// POUs/BACnet Helper/[internal]/_F_BACnet_Utf8ToWin1252
FUNCTION _F_BACnet_Utf8ToWin1252 : BYTE
VAR_INPUT
	pUtf8	: POINTER TO BYTE;
	cbUtf8	: UDINT; (* byte size of UTF8 character (1...6) *)
END_VAR
VAR
	pArr		: POINTER TO ARRAY[0..5] OF BYTE;
	pWord		: POINTER TO ARRAY[0..1] OF BYTE;
	wUCS2		: WORD;
END_VAR
VAR CONSTANT
	cRepl	: BYTE := 16#5F;
END_VAR

(*
	Windows-Codepages
874		Thai
932		Japanisch
936		Vereinfachtes Chinesisch
949		Koreanisch
950		Traditionelles Chinesisch
1250	Mitteleuropäisch
1251	Kyrillisch
1252	Westeuropäisch
1253	Griechisch
1254	Türkisch
1255	Hebräisch
1256	Arabisch
1257	Baltisch
1258	Vietnamesisch
*)
(* first step - convert to UCS2 *)
pArr := pUtf8;
IF (pArr^[0] <= 16#7F) THEN
	(* basic latin *)
	_F_BACnet_Utf8ToWin1252 := pArr^[0];
	RETURN;
ELSIF (cbUtf8 >= 2) THEN
	pWord := ADR(wUCS2);
	IF (pArr^[0] = 16#C2) THEN
		(* latin-1 supplement *)
		wUCS2 := pArr^[1];
	ELSIF (pArr^[0] = 16#C3) AND (pArr^[1] <= 16#BF) THEN
		(* latin-1 supplement *)
		wUCS2 := pArr^[1] + 16#40;
	ELSIF (pArr^[0] = 16#C4) AND (pArr^[1] >= 16#80) THEN
		(* latin extended-A *)
		pWord^[1] := 16#01;
		pWord^[0] := pArr^[1] - 16#80;
	ELSIF (pArr^[0] = 16#C5) AND (pArr^[1] >= 16#80) THEN
		(* latin extended-A *)
		pWord^[1] := 16#01;
		pWord^[0] := pArr^[1] - 16#40;
	ELSIF (pArr^[0] = 16#C6) AND (pArr^[1] >= 16#80) THEN
		(* latin extended-B *)
		pWord^[1] := 16#01;
		pWord^[0] := pArr^[1];
	ELSIF (pArr^[0] = 16#C7) AND (pArr^[1] <= 16#BF) THEN
		(* latin extended-B *)
		pWord^[1] := 16#01;
		pWord^[0] := pArr^[1] + 16#40;
	ELSIF (cbUtf8 >= 3) THEN
		IF (pArr^[0] = 16#E2) AND (pArr^[1] = 16#82) THEN
			(* currency symbols *)
			pWord^[1] := 16#20;
			pWord^[0] := pArr^[2];
		ELSE
			(* unsupported *)
			_F_BACnet_Utf8ToWin1252 := cRepl;
			RETURN;
		END_IF
	ELSE
		(* unsupported *)
		_F_BACnet_Utf8ToWin1252 := cRepl;
		RETURN;
	END_IF
	(* convert UCS2 to Windows-1252 *)
	_F_BACnet_Utf8ToWin1252 := _F_BACnet_UCS2ToWin1252(pWord, FALSE);
	RETURN;
END_IF
(* unsupported *)
_F_BACnet_Utf8ToWin1252 := cRepl;

END_FUNCTION

// POUs/BACnet Helper/[internal]/_F_BACnet_UCS2ToWin1252
FUNCTION _F_BACnet_UCS2ToWin1252 : BYTE
VAR_INPUT
	pUCS2 :	POINTER TO WORD;
	bBE	: BOOL; (* byte-order big endian = TRUE *)
END_VAR
VAR
	pArr : POINTER TO ARRAY[0..1] OF BYTE;
	wUCS2: WORD;
END_VAR
VAR CONSTANT
	cRepl	: BYTE := 16#5F;
END_VAR

(*
	Windows-Codepages
874		Thai
932		Japanisch
936		Vereinfachtes Chinesisch
949		Koreanisch
950		Traditionelles Chinesisch
1250	Mitteleuropäisch
1251	Kyrillisch
1252	Westeuropäisch
1253	Griechisch
1254	Türkisch
1255	Hebräisch
1256	Arabisch
1257	Baltisch
1258	Vietnamesisch
*)
pArr := pUCS2;
IF bBE THEN
	wUCS2 := (pArr^[0] * 16#0100) + pArr^[1];
ELSE
	wUCS2 := pUCS2^;
END_IF
CASE wUCS2 OF
	16#178: 	_F_BACnet_UCS2ToWin1252 := 16#9F;
	16#153: 	_F_BACnet_UCS2ToWin1252 := 16#9C;
	16#152: 	_F_BACnet_UCS2ToWin1252 := 16#8C;
	16#17E: 	_F_BACnet_UCS2ToWin1252 := 16#9E;
	16#17D: 	_F_BACnet_UCS2ToWin1252 := 16#8E;
	16#161: 	_F_BACnet_UCS2ToWin1252 := 16#9A;
	16#160: 	_F_BACnet_UCS2ToWin1252 := 16#8A;
	16#20AC: 	_F_BACnet_UCS2ToWin1252 := 16#80;
	ELSE
		IF wUCS2 <= 16#FF THEN
			_F_BACnet_UCS2ToWin1252 := WORD_TO_BYTE(wUCS2);
		ELSE
			_F_BACnet_UCS2ToWin1252 := cRepl;
		END_IF
END_CASE

END_FUNCTION

// POUs/BACnet Helper/[internal]/_F_BACnet_DecodeUCS2
FUNCTION _F_BACnet_DecodeUCS2 : UDINT (* result is the new character length of the string *)
VAR_INPUT
	pString		: POINTER TO WORD; (* pointer to UCS2 string beginning *)
	cbString	: UDINT; (* byte size of string (use SIZEOF - don't use LEN) *)
END_VAR
VAR
	i		: UDINT;
	pResult	: POINTER TO BYTE;
	pBy		: POINTER TO WORD;
END_VAR

pResult	:= pString;
pBy		:= pString;
FOR i := 0 TO cbString-1 DO
	pResult^ := _F_BACnet_UCS2ToWin1252(pBy, TRUE);
	pBy := pBy + 2;
	(* end-of-string by character *)
	IF (pResult^ = 16#00) THEN
		EXIT;
	END_IF
	(* next character *)
	pResult := pResult + 1;
	(* end-of-string by length *)
	IF (pBy >= (pString + cbString)) THEN
		EXIT;
	END_IF
END_FOR
pResult^ := 16#00;
_F_BACnet_DecodeUCS2 := pResult - pString;

END_FUNCTION

// POUs/BACnet Helper/[internal]/_F_BACnet_DecodeUCS4
FUNCTION _F_BACnet_DecodeUCS4 : UDINT (* result is the new character length of the string *)
VAR_INPUT
	pString		: POINTER TO DWORD; (* pointer to UCS4 string beginning *)
	cbString	: UDINT; (* byte size of string (use SIZEOF - don't use LEN) *)
END_VAR
VAR
	i		: UDINT;
	pResult	: POINTER TO BYTE;
	pBy		: POINTER TO WORD;
END_VAR

pResult	:= pString;
pBy		:= pString;
FOR i := 0 TO cbString-1 DO
	(* byte order big endian *)
	pResult^ := _F_BACnet_UCS2ToWin1252(pBy+2, TRUE);
	pBy := pBy + 4;
	(* end-of-string by character *)
	IF (pResult^ = 16#00) THEN
		EXIT;
	END_IF
	(* next character *)
	pResult := pResult + 1;
	(* end-of-string by length *)
	IF (pBy >= (pString + cbString)) THEN
		EXIT;
	END_IF
END_FOR
pResult^ := 16#00;
_F_BACnet_DecodeUCS4 := pResult - pString;

END_FUNCTION

// POUs/BACnet ADS/Properties/FB_BACnet_EventMessageTextsProperty
FUNCTION_BLOCK FB_BACnet_EventMessageTextsProperty
VAR_INPUT
	tObjectID			: T_BACnet_ObjectIdentifier := 16#FFFFFFFF;
	bAutoGet			: BOOL:=TRUE; (* TRUE = get data from property when ADS connection OR object ID changed *)
	bGet				: BOOL; (* FALSE --> TRUE = get data from property *)
END_VAR
VAR_IN_OUT
	stAdsConn			: ST_BACnet_AdsConnection;
END_VAR
VAR_OUTPUT
	bDone				: BOOL;
	bBusy				: BOOL;
	bError				: BOOL;
	nErrorId			: UINT;
	arrTexts			: ARRAY[0..2] OF T_MaxString; (* Windows-1252 encoded *)
END_VAR
VAR
	_fbReadProp		: FB_BACnet_ReadProp;
	_i				: INT;
	_rtrigGet		: R_TRIG;

	_iEntry			: INT;
	_pEntry			: POINTER TO ST_BACnet_CharacterStringExtListEntry;
	_pText			: POINTER TO BYTE;
	_pByte			: POINTER TO BYTE;
	_bNextEntry		: BOOL;
	_cbEntrySize	: UDINT;
	_cbTmpSize		: UDINT;
	_cbTotalBuf		: UDINT;
	_nAdsReloadOld	: USINT;
	_tObjectIDOld	: T_BACnet_ObjectIdentifier := 16#FFFFFFFF;
	_strExtDecode	: FB_BACnet_StringExtDecode;

END_VAR

(*

Listheader:

typedef struct _ListEntryHdr
{
      DWORD nEntrySize;
      DWORD hdrInfo;
}ListEntryHdr, *PListEntryHdr;


typedef struct _BACnetCharacterString
{
      ULONG       cookie            : 8; // = 0 -> do differentiate normal strings
      ULONG       encoding          : 8; 
      ULONG       strLen            : 16;
      BYTE        stringData[BACNET_STRING_MAXLENGTH];
}BACnetCharacterString, *PBACnetCharacterString;

#define     BACNET_STRING_MAXLENGTH 256

*)

(* ADS read *)
_fbReadProp(
	BACnetDevicePort	:= stAdsConn.nAmsPort,
	bExecute			:= ,
	sNetId				:= stAdsConn.sAmsNetId,
	ObjectType			:= F_BACnet_GetObjType(tObjectID),
	PropertyID			:= BACnetPropertyIdentifier_EventMessageTexts,
	DataType			:= BACnetDataType_CharacterStringExtList,
	ObjectInstance		:= F_BACnet_GetObjInstance(tObjectID),
	ptrValue			:= ADR(stBACnet_AdsBuffer.arrData),
	nLenValue			:= SIZEOF(stBACnet_AdsBuffer.arrData),
	bDone				=> ,
	bBusy				=> ,
	bError				=> ,
	nErrID				=> ,
	nProcessedLen		=> );

(* trigger start event *)
_rtrigGet(CLK:= bGet, Q=> );

(* state machine *)
CASE _i OF

	0: (* Idle *)
		IF 		_rtrigGet.Q
			OR	(		(		(_nAdsReloadOld <> stAdsConn.nReload)
							OR	(_tObjectIDOld <> tObjectID)
						)
					AND	bAutoGet
				)
		THEN
			IF (NOT stAdsConn.bValid) THEN
				(* ADS connection not valid *)
				nErrorId := BACnet_ERR_INVALID_ADS_CONN;
			ELSIF (NOT stAdsConn.bServer AND NOT stAdsConn.bClient) THEN
				(* not a server nor a client *)
				nErrorId := BACnet_ERR_ADS_NoServerClient;
			ELSE
				_i := 1;
				nErrorId := BACnet_ERR_NO_ERROR;
				(* remind parameter *)
				_tObjectIDOld := tObjectID;
				_nAdsReloadOld := stAdsConn.nReload;
			END_IF
			(* reset done flag *)
			bDone := FALSE;
		END_IF
		IF (NOT bGet) AND (NOT bAutoGet) THEN
			nErrorId := BACnet_ERR_NO_ERROR;
			bDone := FALSE;
		END_IF

	(* READ *)
	1: (* read object property data over ADS *)
		IF TestAndSet(stBACnet_AdsBuffer.bTestSet) THEN
			IF _fbReadProp.bExecute THEN
				IF _fbReadProp.bError THEN
					_i := 100;
					nErrorId := BACnet_ERR_ADS_Read;
					_fbReadProp.bExecute := FALSE;
				ELSIF (NOT _fbReadProp.bBusy) THEN
					_i := 2;
					_fbReadProp.bExecute := FALSE;
					_pEntry := ADR(stBACnet_AdsBuffer.arrData);
					MEMSET(ADR(arrTexts), 0, SIZEOF(arrTexts));
					_cbTotalBuf := 0;
					_iEntry := 0;
				END_IF
			ELSE
				(* lock global ADS buffer and start reading *)
				IF stBACnet_AdsBuffer.iLocked = 0 THEN
					_fbReadProp.bExecute := TRUE;
					stBACnet_AdsBuffer.iLocked := SIZEOF(stBACnet_AdsBuffer.arrData);
				END_IF
			END_IF

			(* release temporary task lock *)
			stBACnet_AdsBuffer.bTestSet := FALSE;
		END_IF

	2: (* select time value *)
		WHILE (_i = 2) DO
			_cbEntrySize := _pEntry^.nEntrySize AND 16#7FFFFFFF;
			(* check entry size *)
			IF (_cbEntrySize) > 0 THEN
				(* check index *)
				IF (_iEntry > 2) THEN
					(* error, too many entries *)
					nErrorId := BACnet_ERR_ADS_TooManyEntries;
					_i := 100;
				ELSE
					(* try to decode property data *)
					_strExtDecode(
						pChrStringExt:= ADR(_pEntry^.extString),
						cbOutSize	:= SIZEOF(arrTexts[_iEntry]),
						pOutString	:= ADR(arrTexts[_iEntry]),
						bValid		=> ,
						bOverflow	=> ,
						bUnsupported=> ,
						nLength		=> ,
						eSrcEncoding=> );
					(* check error flags *)
					IF _strExtDecode.bOverflow THEN
						(* text too long *)
						nErrorId := BACnet_ERR_ADS_WrongEntrySize;
						_i := 100;
					ELSIF _strExtDecode.bUnsupported THEN
						(* unsupported encoding *)
						nErrorId := BACnet_ERR_ADS_Encoding;
						_i := 100;
					END_IF
				END_IF
			END_IF

			(* next entry *)
			_NextEntry();
			_iEntry := _iEntry + 1;

			(* check if next entry available *)
			IF (NOT _bNextEntry) THEN
				IF (_iEntry < 3) THEN
					(* not enough entries *)
					nErrorId := BACnet_ERR_ADS_NotEnoughEntries;
				END_IF
				_i := 100;
			END_IF

		END_WHILE

	100: (* Done *)
		bDone := (nErrorId = BACnet_ERR_NO_ERROR);
		(* release ADS buffer *)
		stBACnet_AdsBuffer.iLocked := 0;
		(* go idle *)
		_i := 0;

END_CASE

(* set error flag *)
bError 	:= nErrorId > BACnet_ERR_NO_ERROR;
bBusy 	:= _i > 0;

ACTION _NextEntry:
_bNextEntry := (_pEntry^.nEntrySize AND 16#80000000) = 16#80000000;
_cbTmpSize := _F_BACnet_AlignedSize((_pEntry^.nEntrySize AND 16#7FFFFFFF) + SIZEOF(_pEntry^.nEntrySize) + SIZEOF(_pEntry^.hdrInfo));
_pEntry := _pEntry + _cbTmpSize;
END_ACTION

END_FUNCTION_BLOCK

// POUs/BACnet Helper/[internal]/_F_BACnet_AlignedSize
FUNCTION _F_BACnet_AlignedSize : DWORD
VAR_INPUT
	n	: DWORD;
END_VAR
VAR
END_VAR

_F_BACnet_AlignedSize := (4*(((n)+3)/4));

END_FUNCTION

// POUs/BACnet ADS/Properties/FB_BACnet_ExceptionScheduleProperty
FUNCTION_BLOCK FB_BACnet_ExceptionScheduleProperty
VAR_INPUT
	tObjectID			: T_BACnet_ObjectIdentifier := 16#FFFFFFFF;
	bAutoGet			: BOOL:=TRUE; (* TRUE = get data from property when ADS connection OR object ID changed *)
	bGet				: BOOL; (* FALSE --> TRUE = get data from property *)
	bSet				: BOOL; (* FALSE --> TRUE = set data into property *)
END_VAR
VAR_IN_OUT
	stExceptSched		: ST_BACnet_ExceptionScheduleBool;
	stAdsConn			: ST_BACnet_AdsConnection;
END_VAR
VAR_OUTPUT
	bDone				: BOOL;
	bBusy				: BOOL;
	bError				: BOOL;
	nErrorId			: UINT;
END_VAR
VAR
	_fbReadProp		: FB_BACnet_ReadProp;
	_fbWriteProp	: FB_BACnet_WriteProp;
	_i				: INT;
	_rtrigGet		: R_TRIG;
	_rtrigSet		: R_TRIG;

	_pOldEventEntrySize		: POINTER TO DWORD;
	_pSpEventCalEntryDate	: POINTER TO ST_BACnet_SpecialEventListCalEntryDate;
	_pSpEventCalEntryRange	: POINTER TO ST_BACnet_SpecialEventListCalEntryRange;
	_pSpEventCalEntryWnD	: POINTER TO ST_BACnet_SpecialEventListCalEntryWnD;
	_pSpEventCalRef			: POINTER TO ST_BACnet_SpecialEventListCalReference;
	_pTimeValue		: POINTER TO ST_BACnet_TimeValueList;
	_pOldTimeValue	: POINTER TO ST_BACnet_TimeValueList;

	_iEntry			: INT;
	_iTv			: INT;

	_bNextEvent		: BOOL;
	_bNextTimeValue	: BOOL;

	_cbTmpSize		: UDINT;
	_cbTotalEntry	: UDINT;
	_cbTotalBuf		: UDINT;
	_nAdsReloadOld	: USINT;
	_tObjectIDOld	: T_BACnet_ObjectIdentifier := 16#FFFFFFFF;

END_VAR

(*

Listheader:

typedef struct _ListEntryHdr
{
      DWORD nEntrySize;
      DWORD hdrInfo;
}ListEntryHdr, *PListEntryHdr;

#define ListAlignedSize(n)         (4*(((n)+3)/4))
#define FirstListEntry(p) ( (p)->nEntrySize == 0 )                          ? NULL:p
#define NextListEntry(p) ( ( ((p)->nEntrySize&0x80000000) == 0 ) ? NULL:(PBYTE)(p) + ( ListAlignedSize((p)->nEntrySize&~(0x80000000)) + sizeof(ListEntryHdr)) ) // +4 da für nEntrySize 4 Byte reserviert sind, HighBit ausmaskieren
#define ElemSize(p) ((p)->nEntrySize&(~0x80000000))
#define AlignedEntrySize(p) (ListAlignedSize((p)->nEntrySize&(~0x80000000)))

###################################################################

PropExceptionSchedule:

enum BACnetSpecialEventChoice
{
      calendarEntry,
      calendarReference,
      MaxBACnetSpecialEventChoice
};

typedef struct _BACnetCalendarEntry
{
      BACnetCalendarEntryChoice choice;
      union
      {
            BACnetDate              date;
            BACnetDateRange   dateRange;
            BACnetWeekNDay          weekNDay;
      };
}BACnetCalendarEntry, *PBACnetCalendarEntry;

enum BACnetValueChoice
{
      NullValue                    = 0,
      BoolValue                    = 1,
      UnsignedValue                = 2,
      SignedValue                  = 3,
      RealValue                    = 4,
      DoubleValue                  = 5,
      OctedStringValue        = 6,
      CharStringValue         = 7,
      ObjectIdentifierValue = 8,   // but DataType is 0x0C
      EnumerationValue        = 9,
      MaxBACnetValueChoice    = 10
};

typedef struct _BACnetValue  
{
      BACnetValueChoice choice;
      DWORD                        length;     // Alignment + Datenlänge die folgt
      union
      {
            BOOL                                     boolValue;
            FLOAT                                    realValue;
            DOUBLE                                   doubleValue;
            INT                                      signedValue;
            UINT                                     unsignedValue;
            BYTE*                                    pOctedStringValue; 
            CHAR*                                    pCharStringValue;
            BACnetObjectIdentifier  objectIdentifierValue;
            EnumerationValueType         enumerationValue;
      };
}BACnetValue, *PBACnetValue;

typedef struct _BACnetTimeValue
{
      BACnetTime time;
      DWORD  reserved;  // 64bit Alignment
      BACnetValue value;
}BACnetTimeValue, *PBACnetTimeValue;

typedef struct _BACnetTimeValueList
{
      DWORD nEntrySize; // 0x80000000 -> next entry
      DWORD reserved;
      BACnetTimeValue listEntry;
}BACnetTimeValueList, *PBACnetTimeValueList;

typedef struct _BACnetSpecialEvent
{
      BACnetSpecialEventChoice choice;
      union
      {
            BACnetCalendarEntry calendarEntry;
            BACnetObjectIdentifier calendarReference;
      };
      DWORD eventPriority; // DWORD due to alignment
      DWORD reserved;
      BACnetTimeValueList listOfTimeValues;
}BACnetSpecialEvent, *PBACnetSpecialEvent;

typedef struct _BACnetSpecialEventList
{
      DWORD nEntrySize; // 0x80000000 -> next entry
      DWORD reserved;
      BACnetSpecialEvent listEntry;
}BACnetSpecialEventList, *PBACnetSpecialEventList;

###################################################################

PropWeeklySchedule:

typedef struct _BACnetDailySchedule
{
      DWORD nEntrySize; // 0x80000000 -> next entry
      DWORD reserved;
      BACnetTimeValueList listEntry;
} BACnetDailySchedule, *PBACnetDailySchedule;

###################################################################

PropScheduleDefault / PropPresentValue

typedef struct _BACnetValueList
{
      DWORD nEntrySize; // 0x80000000 -> next entry
      DWORD reserved;
      BACnetValue listEntry;
} BACnetValueList, *PBACnetValueList;

###################################################################

*)

(* ADS read *)
_fbReadProp(
	BACnetDevicePort	:= stAdsConn.nAmsPort,
	bExecute			:= ,
	sNetId				:= stAdsConn.sAmsNetId,
	ObjectType			:= F_BACnet_GetObjType(tObjectID),
	PropertyID			:= BACnetPropertyIdentifier_ExceptionSchedule,
	DataType			:= BACnetDataType_SpecialEventList,
	ObjectInstance		:= F_BACnet_GetObjInstance(tObjectID),
	ptrValue			:= ADR(stBACnet_AdsBuffer.arrData),
	nLenValue			:= SIZEOF(stBACnet_AdsBuffer.arrData),
	bDone				=> ,
	bBusy				=> ,
	bError				=> ,
	nErrID				=> ,
	nProcessedLen		=> );

(* ADS write *)
_fbWriteProp(
	BACnetDevicePort	:= stAdsConn.nAmsPort,
	bExecute			:= ,
	sNetId				:= stAdsConn.sAmsNetId,
	ObjectType			:= F_BACnet_GetObjType(tObjectID),
	PropertyID			:= BACnetPropertyIdentifier_ExceptionSchedule,
	Priority			:= BACnetPriority_None,
	DataType			:= BACnetDataType_SpecialEventList,
	ObjectInstance		:= F_BACnet_GetObjInstance(tObjectID),
	ptrValue			:= ADR(stBACnet_AdsBuffer.arrData),
	nLenValue			:= _cbTotalBuf,
	bDone				=> ,
	bBusy				=> ,
	bError				=> ,
	nErrID				=> );

(* trigger start event *)
_rtrigGet(CLK:= bGet, Q=> );
_rtrigSet(CLK:= bSet, Q=> );

(* state machine *)
CASE _i OF

	0: (* Idle *)
		IF 		_rtrigGet.Q
			OR	_rtrigSet.Q
			OR	(		(		(_nAdsReloadOld <> stAdsConn.nReload)
							OR	(_tObjectIDOld <> tObjectID)
						)
					AND	bAutoGet
				)
			OR	stExceptSched.bReqGet
			OR	stExceptSched.bReqSet
		THEN
			IF (NOT stAdsConn.bValid) THEN
				(* ADS connection not valid *)
				nErrorId := BACnet_ERR_INVALID_ADS_CONN;
			ELSIF (NOT stAdsConn.bServer AND NOT stAdsConn.bClient) THEN
				(* not a server nor a client *)
				nErrorId := BACnet_ERR_ADS_NoServerClient;
			ELSE
				(* decide get or set *)
				IF _rtrigGet.Q OR stExceptSched.bReqGet  THEN
					_i := 1;
					stExceptSched.bReqGet := FALSE;
				ELSIF _rtrigSet.Q OR stExceptSched.bReqSet THEN
					_i := 11;
					stExceptSched.bReqSet := FALSE;
				ELSIF bAutoGet THEN
					_i := 1;
					stExceptSched.bReqGet := FALSE;
				END_IF
				nErrorId := BACnet_ERR_NO_ERROR;
				(* reset index *)
				_iEntry		:= 0;
				(* remind parameter *)
				_tObjectIDOld := tObjectID;
				_nAdsReloadOld := stAdsConn.nReload;
				(* lock data array *)
				stExceptSched.bBusy := TRUE;
			END_IF
			(* reset done flag *)
			bDone := FALSE;
		END_IF
		IF (NOT bGet) AND (NOT bSet) AND (NOT bAutoGet) THEN
			nErrorId := BACnet_ERR_NO_ERROR;
			bDone := FALSE;
		END_IF

	(* READ *)
	1: (* read object property data via ADS *)
		IF TestAndSet(stBACnet_AdsBuffer.bTestSet) THEN
			IF _fbReadProp.bExecute THEN
				IF _fbReadProp.bError THEN
					_i := 100;
					nErrorId := BACnet_ERR_ADS_Read;
					_fbReadProp.bExecute := FALSE;
				ELSIF (NOT _fbReadProp.bBusy) THEN
					_i := 2;
					_fbReadProp.bExecute := FALSE;
					(* prepare pointer *)
					_pSpEventCalEntryDate	:= ADR(stBACnet_AdsBuffer.arrData);
					_pSpEventCalEntryRange	:= ADR(stBACnet_AdsBuffer.arrData);
					_pSpEventCalEntryWnD	:= ADR(stBACnet_AdsBuffer.arrData);
					_pSpEventCalRef			:= ADR(stBACnet_AdsBuffer.arrData);
					(* clear output data *)
					MEMSET(ADR(stExceptSched.arrEntries), 0, SIZEOF(stExceptSched.arrEntries));
					_cbTotalBuf := 0;
					_bNextEvent := TRUE;
				END_IF

			ELSIF (stBACnet_AdsBuffer.iLocked = 0) THEN
				_fbReadProp.bExecute := TRUE;
				(* lock global ADS buffer *)
				stBACnet_AdsBuffer.iLocked := SIZEOF(stBACnet_AdsBuffer.arrData);
			END_IF

			(* release temporary task lock *)
			stBACnet_AdsBuffer.bTestSet := FALSE;
		END_IF

	2: (* select event entry *)
		(* more events? *)
		IF (NOT _bNextEvent) THEN
			(* no more events, exit *)
			_i := 4;
		ELSE
			_i := 3;
			(* check if local buffer is full *)
			IF _iEntry > to_int(BACnet_MaxExSchEntries) THEN
				_i := 4; (* maximum entries reached --> finished *)
			ELSIF ((_pSpEventCalEntryDate^.nEntrySize AND 16#7FFFFFFF) > 0) THEN
				(* initialize first entry *)
				stExceptSched.arrEntries[_iEntry].eEntryType := BACnetCalendarEntryType_None;

				CASE _pSpEventCalEntryDate^.stListEntry.eEventChoice OF

					BACnetSpecialEventChoice_calendarReference:
						_pTimeValue := ADR(_pSpEventCalRef^.stListEntry.stListOfTimeValues);
						stExceptSched.arrEntries[_iEntry].eEntryType := BACnetCalendarEntryType_Ref;
						stExceptSched.arrEntries[_iEntry].stCalRef.tCalObjectId := _pSpEventCalRef^.stListEntry.tCalRef;
						stExceptSched.arrEntries[_iEntry].ePriority := DWORD_TO_INT(_pSpEventCalRef^.stListEntry.iEventPriority);

					BACnetSpecialEventChoice_calendarEntry:
						CASE _pSpEventCalEntryDate^.stListEntry.stCalEntry.eEntryChoice OF
							BACnetCalendarEntryChoice_date:
								_pTimeValue := ADR(_pSpEventCalEntryDate^.stListEntry.stListOfTimeValues);
								stExceptSched.arrEntries[_iEntry].eEntryType := BACnetCalendarEntryType_Date;
								stExceptSched.arrEntries[_iEntry].stDate.stStart := _pSpEventCalEntryDate^.stListEntry.stCalEntry.stDate;
								stExceptSched.arrEntries[_iEntry].stDate.stEnd := _pSpEventCalEntryDate^.stListEntry.stCalEntry.stDate;
								stExceptSched.arrEntries[_iEntry].ePriority := DWORD_TO_INT(_pSpEventCalEntryDate^.stListEntry.iEventPriority);

							BACnetCalendarEntryChoice_dateRange:
								_pTimeValue := ADR(_pSpEventCalEntryRange^.stListEntry.stListOfTimeValues);
								stExceptSched.arrEntries[_iEntry].eEntryType := BACnetCalendarEntryType_DateRange;
								stExceptSched.arrEntries[_iEntry].stDate.stStart := _pSpEventCalEntryRange^.stListEntry.stCalEntry.stStartDate;
								stExceptSched.arrEntries[_iEntry].stDate.stEnd := _pSpEventCalEntryRange^.stListEntry.stCalEntry.stEndDate;
								stExceptSched.arrEntries[_iEntry].ePriority := DWORD_TO_INT(_pSpEventCalEntryRange^.stListEntry.iEventPriority);

							BACnetCalendarEntryChoice_weekNDay:
								_pTimeValue := ADR(_pSpEventCalEntryWnD^.stListEntry.stListOfTimeValues);
								stExceptSched.arrEntries[_iEntry].eEntryType := BACnetCalendarEntryType_WeekNDay;
								stExceptSched.arrEntries[_iEntry].stWeekNDay.iMonth := _pSpEventCalEntryWnD^.stListEntry.stCalEntry.iMonth;
								stExceptSched.arrEntries[_iEntry].stWeekNDay.iWeekOfMonth := _pSpEventCalEntryWnD^.stListEntry.stCalEntry.iWeekOfMonth;
								stExceptSched.arrEntries[_iEntry].stWeekNDay.iDay := _pSpEventCalEntryWnD^.stListEntry.stCalEntry.iDay;
								stExceptSched.arrEntries[_iEntry].ePriority := DWORD_TO_INT(_pSpEventCalEntryWnD^.stListEntry.iEventPriority);

							ELSE
								(* unknown entry choice *)
								nErrorId := BACnet_ERR_UnknownEntryChoice;
								_i := 100;
						END_CASE
					ELSE
						(* unknown event choice *)
						nErrorId := BACnet_ERR_UnknownEventChoice;
						_i := 100;
				END_CASE
			ELSE
				(* mark as invalid *)
				stExceptSched.arrEntries[_iEntry].eEntryType := BACnetCalendarEntryType_None;
			END_IF
		END_IF
		(* reset time value index *)
		_iTv := 0;

	3: (* scan time value list *)
		(* preset next time value flag *)
		_bNextTimeValue := TRUE;
		(* loop till all time values are parsed *)
		WHILE _bNextTimeValue AND _pTimeValue <> 0 DO
			IF ((_pTimeValue^.nEntrySize AND 16#7FFFFFFF) > 0) AND (_iTv <= TO_INT(BACnet_MaxTimeValues)) THEN
				(* time value data available - is it a bool type? *)
				IF		_pTimeValue^.stListEntry.stValue.eValueChoice = BACnetDataType_Bool
					OR	_pTimeValue^.stListEntry.stValue.eValueChoice = BACnetDataType_Null
				THEN
					(* decide entry type *)
					CASE stExceptSched.arrEntries[_iEntry].eEntryType OF
						BACnetCalendarEntryType_Date,
						BACnetCalendarEntryType_DateRange:
							stExceptSched.arrEntries[_iEntry].arrTimeValue[_iTv].bValid := TRUE;
							stExceptSched.arrEntries[_iEntry].arrTimeValue[_iTv].stTime := _pTimeValue^.stListEntry.stTime;
							stExceptSched.arrEntries[_iEntry].arrTimeValue[_iTv].eType := _pTimeValue^.stListEntry.stValue.eValueChoice;
							IF _pTimeValue^.stListEntry.stValue.cbData = 1 THEN
								MEMCPY(	ADR(stExceptSched.arrEntries[_iEntry].arrTimeValue[_iTv].bValue),
										ADR(_pTimeValue^.stListEntry.stValue.nData),
										SIZEOF(stExceptSched.arrEntries[_iEntry].arrTimeValue[_iTv].bValue)
								);
							ELSE
								stExceptSched.arrEntries[_iEntry].arrTimeValue[_iTv].bValue := FALSE;
							END_IF
							_iTv := _iTv +1;

						BACnetCalendarEntryType_WeekNDay:
							stExceptSched.arrEntries[_iEntry].arrTimeValue[_iTv].bValid := TRUE;
							stExceptSched.arrEntries[_iEntry].arrTimeValue[_iTv].stTime := _pTimeValue^.stListEntry.stTime;
							stExceptSched.arrEntries[_iEntry].arrTimeValue[_iTv].eType := _pTimeValue^.stListEntry.stValue.eValueChoice;
							IF _pTimeValue^.stListEntry.stValue.cbData = 1 THEN
								MEMCPY(	ADR(stExceptSched.arrEntries[_iEntry].arrTimeValue[_iTv].bValue),
										ADR(_pTimeValue^.stListEntry.stValue.nData),
										SIZEOF(stExceptSched.arrEntries[_iEntry].arrTimeValue[_iTv].bValue)
								);
							ELSE
								stExceptSched.arrEntries[_iEntry].arrTimeValue[_iTv].bValue := FALSE;
							END_IF
							_iTv := _iTv +1;

						BACnetCalendarEntryType_Ref:
							stExceptSched.arrEntries[_iEntry].arrTimeValue[_iTv].bValid := TRUE;
							stExceptSched.arrEntries[_iEntry].arrTimeValue[_iTv].stTime := _pTimeValue^.stListEntry.stTime;
							stExceptSched.arrEntries[_iEntry].arrTimeValue[_iTv].eType := _pTimeValue^.stListEntry.stValue.eValueChoice;
							IF _pTimeValue^.stListEntry.stValue.cbData = 1 THEN
								MEMCPY(	ADR(stExceptSched.arrEntries[_iEntry].arrTimeValue[_iTv].bValue),
										ADR(_pTimeValue^.stListEntry.stValue.nData),
										SIZEOF(stExceptSched.arrEntries[_iEntry].arrTimeValue[_iTv].bValue)
								);
							ELSE
								stExceptSched.arrEntries[_iEntry].arrTimeValue[_iTv].bValue := FALSE;
							END_IF
							_iTv := _iTv +1;

					END_CASE

				ELSE
					(* unsupported data type *);
				END_IF

			END_IF

			(* empty entry size or data buffer full, next time value entry *)
			_NextTimeValue();

		END_WHILE

		(* count *)(*
		IF _iTv > 0 THEN
			_iEntry := _iEntry +1;
		END_IF*)
		_iEntry := _iEntry +1;

		(* next event entry *)
		_NextEvent();
		_i := 2;

	4: (* data read and parsed successful *)
		stExceptSched.nGet := stExceptSched.nGet +1;
		_i := 100;

	11: (* lock global ADS buffer *)
		IF TestAndSet(stBACnet_AdsBuffer.bTestSet) THEN
			IF stBACnet_AdsBuffer.iLocked = 0 THEN
				stBACnet_AdsBuffer.iLocked := SIZEOF(stBACnet_AdsBuffer.arrData);
				(* initalize total size counter *)
				_cbTotalBuf := 0;
				(* prepare pointer *)
				_pSpEventCalEntryDate	:= ADR(stBACnet_AdsBuffer.arrData);
				_pSpEventCalEntryRange	:= ADR(stBACnet_AdsBuffer.arrData);
				_pSpEventCalEntryWnD	:= ADR(stBACnet_AdsBuffer.arrData);
				_pSpEventCalRef			:= ADR(stBACnet_AdsBuffer.arrData);
				_pOldEventEntrySize		:= 0;
				(* loop against input data *)
				_i := 12;
			END_IF
			(* release temporary task lock *)
			stBACnet_AdsBuffer.bTestSet := FALSE;
		END_IF

	12: (* write calendar entries date/date range *)
		FOR _iEntry := 0 TO TO_INT(BACnet_MaxExSchEntries) DO

			_pOldTimeValue	:= 0;
			_cbTotalEntry	:= 0;

			IF stExceptSched.arrEntries[_iEntry].eEntryType <> BACnetCalendarEntryType_None THEN
				(* valid entry *)
				CASE stExceptSched.arrEntries[_iEntry].eEntryType OF

					BACnetCalendarEntryType_Date,
					BACnetCalendarEntryType_DateRange:
						(* set special entry choice *)
						IF stExceptSched.arrEntries[_iEntry].eEntryType = BACnetCalendarEntryType_Date THEN
							_pSpEventCalEntryDate^.stListEntry.eEventChoice := BACnetSpecialEventChoice_calendarEntry;
							_pSpEventCalEntryDate^.stListEntry.nRes1 := 0;
							(* set time value pointer *)
							_pTimeValue := ADR(_pSpEventCalEntryDate^.stListEntry.stListOfTimeValues);
						ELSE
							_pSpEventCalEntryRange^.stListEntry.eEventChoice := BACnetSpecialEventChoice_calendarEntry;
							_pSpEventCalEntryRange^.stListEntry.nRes1 := 0;
							(* set time value pointer *)
							_pTimeValue := ADR(_pSpEventCalEntryRange^.stListEntry.stListOfTimeValues);
						END_IF

					BACnetCalendarEntryType_WeekNDay:
						(* set special entry choice *)
						_pSpEventCalEntryWnD^.stListEntry.eEventChoice := BACnetSpecialEventChoice_calendarEntry;
						_pSpEventCalEntryWnD^.stListEntry.nRes1 := 0;
						(* set time value pointer *)
						_pTimeValue := ADR(_pSpEventCalEntryWnD^.stListEntry.stListOfTimeValues);

					BACnetCalendarEntryType_Ref:
						(* set special entry choice *)
						_pSpEventCalRef^.stListEntry.eEventChoice := BACnetSpecialEventChoice_calendarReference;
						_pSpEventCalRef^.stListEntry.nRes1 := 0;
						(* set time value pointer *)
						_pTimeValue := ADR(_pSpEventCalRef^.stListEntry.stListOfTimeValues);

				END_CASE


				(* loop against time values *)
				FOR _iTv := 0 TO TO_INT(BACnet_MaxTimeValues) DO

					(* valid entry? *)
					IF stExceptSched.arrEntries[_iEntry].arrTimeValue[_iTv].bValid THEN
						(* copy time *)
						_pTimeValue^.stListEntry.stTime := stExceptSched.arrEntries[_iEntry].arrTimeValue[_iTv].stTime;
						_pTimeValue^.stListEntry.stValue.nData := 0; (* clear data *)
						(* decide between None and Bool type *)
						IF stExceptSched.arrEntries[_iEntry].arrTimeValue[_iTv].eType = BACnetDataType_Bool THEN
							(* BOOL type *)
							_pTimeValue^.stListEntry.stValue.eValueChoice := BACnetDataType_Bool;
							_pTimeValue^.stListEntry.stValue.nRes1 := 0;
							_pTimeValue^.stListEntry.stValue.cbData := SIZEOF(stExceptSched.arrEntries[_iEntry].arrTimeValue[_iTv].bValue);
							MEMCPY(	ADR(_pTimeValue^.stListEntry.stValue.nData),
									ADR(stExceptSched.arrEntries[_iEntry].arrTimeValue[_iTv].bValue),
									MIN(SIZEOF(_pTimeValue^.stListEntry.stValue.nData), _pTimeValue^.stListEntry.stValue.cbData)
							);
						ELSE
							(* other or NONE type *)
							_pTimeValue^.stListEntry.stValue.eValueChoice := BACnetDataType_Null;
							_pTimeValue^.stListEntry.stValue.nRes1 := 0;
							_pTimeValue^.stListEntry.stValue.cbData := 0;
						END_IF

						(* calculate time-value entry size *)
						_pTimeValue^.nEntrySize :=	_pTimeValue^.stListEntry.stValue.cbData
												+	SIZEOF(_pTimeValue^.stListEntry.nRes)
												+	SIZEOF(_pTimeValue^.stListEntry.stTime)
												+	SIZEOF(_pTimeValue^.stListEntry.stValue.cbData)
												+	SIZEOF(_pTimeValue^.stListEntry.stValue.eValueChoice)
												+	SIZEOF(_pTimeValue^.stListEntry.stValue.nRes1);

						IF (_iTv > 0 AND _pOldTimeValue <> 0) THEN
							(* next entry flag *)
							_pOldTimeValue^.nEntrySize := _pOldTimeValue^.nEntrySize + 16#80000000;
						END_IF

						(* update time value pointer *)
						_NextTimeValue();

						(* ...and add to total entry size counter *)
						_cbTotalEntry := _cbTotalEntry + _cbTmpSize;

					ELSE
						(* clear entry *)
						_pTimeValue^.nEntrySize := 0;
						_pTimeValue^.stListEntry.stValue.cbData := 0;
					END_IF

				END_FOR

				(* check if time value list is empty *)
				IF _cbTotalEntry = 0 THEN
					(* no time values, set default size *)
					_cbTotalEntry := SIZEOF(_pTimeValue^.nEntrySize) + SIZEOF(_pTimeValue^.nRes);
				END_IF

				(* caclulate event entry size *)
				CASE stExceptSched.arrEntries[_iEntry].eEntryType OF

					BACnetCalendarEntryType_Date:
						(* caclulate event entry size and write into data structure *)
						_pSpEventCalEntryDate^.nEntrySize :=	_cbTotalEntry
															+	SIZEOF(_pSpEventCalEntryDate^.stListEntry.eEventChoice)
															+	SIZEOF(_pSpEventCalEntryDate^.stListEntry.iEventPriority)
															+	SIZEOF(_pSpEventCalEntryDate^.stListEntry.nRes1)
															+	SIZEOF(_pSpEventCalEntryDate^.stListEntry.nRes2)
															+	SIZEOF(_pSpEventCalEntryDate^.stListEntry.nRes3)
															+	SIZEOF(_pSpEventCalEntryDate^.stListEntry.stCalEntry);
						(* copy event data *)
						_pSpEventCalEntryDate^.stListEntry.eEventChoice := BACnetSpecialEventChoice_calendarEntry;
						_pSpEventCalEntryDate^.stListEntry.nRes1 := 0;
						_pSpEventCalEntryDate^.stListEntry.iEventPriority := to_dword(stExceptSched.arrEntries[_iEntry].ePriority);
						_pSpEventCalEntryDate^.stListEntry.stCalEntry.eEntryChoice := BACnetCalendarEntryChoice_date;
						_pSpEventCalEntryDate^.stListEntry.stCalEntry.nRes := 0;
						_pSpEventCalEntryDate^.stListEntry.stCalEntry.stDate := stExceptSched.arrEntries[_iEntry].stDate.stStart;

					BACnetCalendarEntryType_DateRange:
						(* caclulate event entry size and write into data structure *)
						_pSpEventCalEntryRange^.nEntrySize :=	_cbTotalEntry
															+	SIZEOF(_pSpEventCalEntryRange^.stListEntry.eEventChoice)
															+	SIZEOF(_pSpEventCalEntryRange^.stListEntry.iEventPriority)
															+	SIZEOF(_pSpEventCalEntryRange^.stListEntry.nRes1)
															+	SIZEOF(_pSpEventCalEntryRange^.stListEntry.nRes2)
															+	SIZEOF(_pSpEventCalEntryRange^.stListEntry.stCalEntry);
						(* copy event data *)
						_pSpEventCalEntryRange^.stListEntry.eEventChoice := BACnetSpecialEventChoice_calendarEntry;
						_pSpEventCalEntryRange^.stListEntry.nRes1 := 0;
						_pSpEventCalEntryRange^.stListEntry.iEventPriority := TO_DWORD(stExceptSched.arrEntries[_iEntry].ePriority);
						_pSpEventCalEntryRange^.stListEntry.stCalEntry.eEntryChoice := BACnetCalendarEntryChoice_dateRange;
						_pSpEventCalEntryRange^.stListEntry.stCalEntry.nRes := 0;
						_pSpEventCalEntryRange^.stListEntry.stCalEntry.stStartDate := stExceptSched.arrEntries[_iEntry].stDate.stStart;
						_pSpEventCalEntryRange^.stListEntry.stCalEntry.stEndDate := stExceptSched.arrEntries[_iEntry].stDate.stEnd;

					BACnetCalendarEntryType_WeekNDay:
						(* caclulate event entry size and write into data structure *)
						_pSpEventCalEntryWnD^.nEntrySize :=	_cbTotalEntry
															+	SIZEOF(_pSpEventCalEntryWnD^.stListEntry.eEventChoice)
															+	SIZEOF(_pSpEventCalEntryWnD^.stListEntry.iEventPriority)
															+	SIZEOF(_pSpEventCalEntryWnD^.stListEntry.nRes1)
															+	SIZEOF(_pSpEventCalEntryWnD^.stListEntry.nRes2)
															+	SIZEOF(_pSpEventCalEntryWnD^.stListEntry.nRes3)
															+	SIZEOF(_pSpEventCalEntryWnD^.stListEntry.stCalEntry);
						(* copy event data *)
						_pSpEventCalEntryWnD^.stListEntry.eEventChoice := BACnetSpecialEventChoice_calendarEntry;
						_pSpEventCalEntryWnD^.stListEntry.nRes1 := 0;
						_pSpEventCalEntryWnD^.stListEntry.iEventPriority := to_dword(stExceptSched.arrEntries[_iEntry].ePriority);
						_pSpEventCalEntryWnD^.stListEntry.stCalEntry.eEntryChoice := BACnetCalendarEntryChoice_weekNDay;
						_pSpEventCalEntryWnD^.stListEntry.stCalEntry.nRes1 := 0;
						_pSpEventCalEntryWnD^.stListEntry.stCalEntry.iDay := stExceptSched.arrEntries[_iEntry].stWeekNDay.iDay;
						_pSpEventCalEntryWnD^.stListEntry.stCalEntry.iMonth := stExceptSched.arrEntries[_iEntry].stWeekNDay.iMonth;
						_pSpEventCalEntryWnD^.stListEntry.stCalEntry.iWeekOfMonth := stExceptSched.arrEntries[_iEntry].stWeekNDay.iWeekOfMonth;

					BACnetCalendarEntryType_Ref:
						(* caclulate event entry size and write into data structure *)
						_pSpEventCalRef^.nEntrySize :=	_cbTotalEntry
													+	SIZEOF(_pSpEventCalRef^.stListEntry.eEventChoice)
													+	SIZEOF(_pSpEventCalRef^.stListEntry.iEventPriority)
													+	SIZEOF(_pSpEventCalRef^.stListEntry.nRes1)
													+	SIZEOF(_pSpEventCalRef^.stListEntry.nRes2)
													+	SIZEOF(_pSpEventCalRef^.stListEntry.nRes3)
													+	SIZEOF(_pSpEventCalRef^.stListEntry.nRes4)
													+	SIZEOF(_pSpEventCalRef^.stListEntry.tCalRef);
						(* copy event data *)
						_pSpEventCalRef^.stListEntry.eEventChoice := BACnetSpecialEventChoice_calendarReference;
						_pSpEventCalRef^.stListEntry.nRes1 := 0;
						_pSpEventCalRef^.stListEntry.iEventPriority := to_dword(stExceptSched.arrEntries[_iEntry].ePriority);
						_pSpEventCalRef^.stListEntry.tCalRef := stExceptSched.arrEntries[_iEntry].stCalRef.tCalObjectId;

				END_CASE

				(* set next entry flag *)
				IF (_pOldEventEntrySize <> 0) THEN
					_pOldEventEntrySize^ := _pOldEventEntrySize^ + 16#80000000;
				END_IF

				(* next calendar entry *)
				_NextEvent();
			END_IF

		END_FOR

		(* send data *)
		_i := 19;

	19:
		IF _fbWriteProp.bExecute AND (NOT _fbWriteProp.bBusy) THEN
			(* check result *)
			_fbWriteProp.bExecute := FALSE;
			IF _fbWriteProp.bError THEN
				nErrorId := BACnet_ERR_ADS_Write;
			ELSE
				stExceptSched.nSet := stExceptSched.nSet +1;
			END_IF
			_i := 100;
		ELSE
			(* start ADS write *)
			_fbWriteProp.bExecute := TRUE;
		END_IF

	100: (* Done *)
		bDone := (nErrorId = BACnet_ERR_NO_ERROR);
		(* release ADS buffer *)
		stBACnet_AdsBuffer.iLocked := 0;
		(* release data array *)
		stExceptSched.bBusy := FALSE;
		(* go idle *)
		_i := 0;

END_CASE

(* set error flag *)
bError 	:= nErrorId > BACnet_ERR_NO_ERROR;
bBusy 	:= _i > 0;

ACTION _NextEvent:
_bNextEvent := ((_pSpEventCalEntryDate^.nEntrySize AND 16#80000000) = 16#80000000);
_cbTmpSize := _F_BACnet_AlignedSize(_pSpEventCalEntryDate^.nEntrySize AND 16#7FFFFFFF) + SIZEOF(_pSpEventCalEntryDate^.nEntrySize) + SIZEOF(_pSpEventCalEntryDate^.nRes);
_pOldEventEntrySize		:= ADR(_pSpEventCalEntryDate^.nEntrySize);
_pSpEventCalEntryDate	:= _pSpEventCalEntryDate + _cbTmpSize;
_pSpEventCalEntryRange	:= _pSpEventCalEntryRange + _cbTmpSize;
_pSpEventCalEntryWnD	:= _pSpEventCalEntryWnD + _cbTmpSize;
_pSpEventCalRef			:= _pSpEventCalRef + _cbTmpSize;
_cbTotalBuf := _cbTotalBuf + _cbTmpSize;
_pOldTimeValue := 0;
END_ACTION

ACTION _NextTimeValue:
_bNextTimeValue := (_pTimeValue^.nEntrySize AND 16#80000000) = 16#80000000;
_cbTmpSize := 	(_F_BACnet_AlignedSize(_pTimeValue^.nEntrySize) AND 16#7FFFFFFF)
			+	SIZEOF(_pTimeValue^.nEntrySize)
			+	SIZEOF(_pTimeValue^.nRes);
_pOldTimeValue := _pTimeValue;
_pTimeValue := _pTimeValue + _cbTmpSize;
END_ACTION

END_FUNCTION_BLOCK

// POUs/BACnet ADS/Properties/FB_BACnet_ExceptionSchedulePropertyReal
FUNCTION_BLOCK FB_BACnet_ExceptionSchedulePropertyReal
VAR_INPUT
	tObjectID			: T_BACnet_ObjectIdentifier := 16#FFFFFFFF;
	bAutoGet			: BOOL:=TRUE; (* TRUE = get data from property when ADS connection OR object ID changed *)
	bGet				: BOOL; (* FALSE --> TRUE = get data from property *)
	bSet				: BOOL; (* FALSE --> TRUE = set data into property *)
END_VAR
VAR_IN_OUT
	stExceptSched		: ST_BACnet_ExceptionScheduleReal;
	stAdsConn			: ST_BACnet_AdsConnection;
END_VAR
VAR_OUTPUT
	bDone				: BOOL;
	bBusy				: BOOL;
	bError				: BOOL;
	nErrorId			: UINT;
END_VAR
VAR
	_fbReadProp		: FB_BACnet_ReadProp;
	_fbWriteProp	: FB_BACnet_WriteProp;
	_i				: INT;
	_rtrigGet		: R_TRIG;
	_rtrigSet		: R_TRIG;

	_pOldEventEntrySize		: POINTER TO DWORD;
	_pSpEventCalEntryDate	: POINTER TO ST_BACnet_SpecialEventListCalEntryDate;
	_pSpEventCalEntryRange	: POINTER TO ST_BACnet_SpecialEventListCalEntryRange;
	_pSpEventCalEntryWnD	: POINTER TO ST_BACnet_SpecialEventListCalEntryWnD;
	_pSpEventCalRef			: POINTER TO ST_BACnet_SpecialEventListCalReference;
	_pTimeValue		: POINTER TO ST_BACnet_TimeValueList;
	_pOldTimeValue	: POINTER TO ST_BACnet_TimeValueList;

	_iEntry			: INT;
	_iTv			: INT;

	_bNextEvent		: BOOL;
	_bNextTimeValue	: BOOL;

	_cbTmpSize		: UDINT;
	_cbTotalEntry	: UDINT;
	_cbTotalBuf		: UDINT;
	_nAdsReloadOld	: USINT;
	_tObjectIDOld	: T_BACnet_ObjectIdentifier := 16#FFFFFFFF;

	_pReal			: POINTER TO REAL;
END_VAR

(*

Listheader:

typedef struct _ListEntryHdr
{
      DWORD nEntrySize;
      DWORD hdrInfo;
}ListEntryHdr, *PListEntryHdr;

#define ListAlignedSize(n)         (4*(((n)+3)/4))
#define FirstListEntry(p) ( (p)->nEntrySize == 0 )                          ? NULL:p
#define NextListEntry(p) ( ( ((p)->nEntrySize&0x80000000) == 0 ) ? NULL:(PBYTE)(p) + ( ListAlignedSize((p)->nEntrySize&~(0x80000000)) + sizeof(ListEntryHdr)) ) // +4 da für nEntrySize 4 Byte reserviert sind, HighBit ausmaskieren
#define ElemSize(p) ((p)->nEntrySize&(~0x80000000))
#define AlignedEntrySize(p) (ListAlignedSize((p)->nEntrySize&(~0x80000000)))

###################################################################

PropExceptionSchedule:

enum BACnetSpecialEventChoice
{
      calendarEntry,
      calendarReference,
      MaxBACnetSpecialEventChoice
};

typedef struct _BACnetCalendarEntry
{
      BACnetCalendarEntryChoice choice;
      union
      {
            BACnetDate              date;
            BACnetDateRange   dateRange;
            BACnetWeekNDay          weekNDay;
      };
}BACnetCalendarEntry, *PBACnetCalendarEntry;

enum BACnetValueChoice
{
      NullValue                    = 0,
      BoolValue                    = 1,
      UnsignedValue                = 2,
      SignedValue                  = 3,
      RealValue                    = 4,
      DoubleValue                  = 5,
      OctedStringValue        = 6,
      CharStringValue         = 7,
      ObjectIdentifierValue = 8,   // but DataType is 0x0C
      EnumerationValue        = 9,
      MaxBACnetValueChoice    = 10
};

typedef struct _BACnetValue  
{
      BACnetValueChoice choice;
      DWORD                        length;     // Alignment + Datenlänge die folgt
      union
      {
            BOOL                                     boolValue;
            FLOAT                                    realValue;
            DOUBLE                                   doubleValue;
            INT                                      signedValue;
            UINT                                     unsignedValue;
            BYTE*                                    pOctedStringValue; 
            CHAR*                                    pCharStringValue;
            BACnetObjectIdentifier  objectIdentifierValue;
            EnumerationValueType         enumerationValue;
      };
}BACnetValue, *PBACnetValue;

typedef struct _BACnetTimeValue
{
      BACnetTime time;
      DWORD  reserved;  // 64bit Alignment
      BACnetValue value;
}BACnetTimeValue, *PBACnetTimeValue;

typedef struct _BACnetTimeValueList
{
      DWORD nEntrySize; // 0x80000000 -> next entry
      DWORD reserved;
      BACnetTimeValue listEntry;
}BACnetTimeValueList, *PBACnetTimeValueList;

typedef struct _BACnetSpecialEvent
{
      BACnetSpecialEventChoice choice;
      union
      {
            BACnetCalendarEntry calendarEntry;
            BACnetObjectIdentifier calendarReference;
      };
      DWORD eventPriority; // DWORD due to alignment
      DWORD reserved;
      BACnetTimeValueList listOfTimeValues;
}BACnetSpecialEvent, *PBACnetSpecialEvent;

typedef struct _BACnetSpecialEventList
{
      DWORD nEntrySize; // 0x80000000 -> next entry
      DWORD reserved;
      BACnetSpecialEvent listEntry;
}BACnetSpecialEventList, *PBACnetSpecialEventList;

###################################################################

PropWeeklySchedule:

typedef struct _BACnetDailySchedule
{
      DWORD nEntrySize; // 0x80000000 -> next entry
      DWORD reserved;
      BACnetTimeValueList listEntry;
} BACnetDailySchedule, *PBACnetDailySchedule;

###################################################################

PropScheduleDefault / PropPresentValue

typedef struct _BACnetValueList
{
      DWORD nEntrySize; // 0x80000000 -> next entry
      DWORD reserved;
      BACnetValue listEntry;
} BACnetValueList, *PBACnetValueList;

###################################################################

*)

(* ADS read *)
_fbReadProp(
	BACnetDevicePort	:= stAdsConn.nAmsPort,
	bExecute			:= ,
	sNetId				:= stAdsConn.sAmsNetId,
	ObjectType			:= F_BACnet_GetObjType(tObjectID),
	PropertyID			:= BACnetPropertyIdentifier_ExceptionSchedule,
	DataType			:= BACnetDataType_SpecialEventList,
	ObjectInstance		:= F_BACnet_GetObjInstance(tObjectID),
	ptrValue			:= ADR(stBACnet_AdsBuffer.arrData),
	nLenValue			:= SIZEOF(stBACnet_AdsBuffer.arrData),
	bDone				=> ,
	bBusy				=> ,
	bError				=> ,
	nErrID				=> ,
	nProcessedLen		=> );

(* ADS write *)
_fbWriteProp(
	BACnetDevicePort	:= stAdsConn.nAmsPort,
	bExecute			:= ,
	sNetId				:= stAdsConn.sAmsNetId,
	ObjectType			:= F_BACnet_GetObjType(tObjectID),
	PropertyID			:= BACnetPropertyIdentifier_ExceptionSchedule,
	Priority			:= BACnetPriority_None,
	DataType			:= BACnetDataType_SpecialEventList,
	ObjectInstance		:= F_BACnet_GetObjInstance(tObjectID),
	ptrValue			:= ADR(stBACnet_AdsBuffer.arrData),
	nLenValue			:= _cbTotalBuf,
	bDone				=> ,
	bBusy				=> ,
	bError				=> ,
	nErrID				=> );

(* trigger start event *)
_rtrigGet(CLK:= bGet, Q=> );
_rtrigSet(CLK:= bSet, Q=> );

(* state machine *)
CASE _i OF

	0: (* Idle *)
		IF 		_rtrigGet.Q
			OR	_rtrigSet.Q
			OR	(		(		(_nAdsReloadOld <> stAdsConn.nReload)
							OR	(_tObjectIDOld <> tObjectID)
						)
					AND	bAutoGet
				)
			OR	stExceptSched.bReqGet
			OR	stExceptSched.bReqSet
		THEN
			IF (NOT stAdsConn.bValid) THEN
				(* ADS connection not valid *)
				nErrorId := BACnet_ERR_INVALID_ADS_CONN;
			ELSIF (NOT stAdsConn.bServer AND NOT stAdsConn.bClient) THEN
				(* not a server nor a client *)
				nErrorId := BACnet_ERR_ADS_NoServerClient;
			ELSE
				(* decide get or set *)
				IF _rtrigGet.Q OR stExceptSched.bReqGet  THEN
					_i := 1;
					stExceptSched.bReqGet := FALSE;
				ELSIF _rtrigSet.Q OR stExceptSched.bReqSet THEN
					_i := 11;
					stExceptSched.bReqSet := FALSE;
				ELSIF bAutoGet THEN
					_i := 1;
					stExceptSched.bReqGet := FALSE;
				END_IF
				nErrorId := BACnet_ERR_NO_ERROR;
				(* reset index *)
				_iEntry		:= 0;
				(* remind parameter *)
				_tObjectIDOld := tObjectID;
				_nAdsReloadOld := stAdsConn.nReload;
				(* lock data array *)
				stExceptSched.bBusy := TRUE;
			END_IF
			(* reset done flag *)
			bDone := FALSE;
		END_IF
		IF (NOT bGet) AND (NOT bSet) AND (NOT bAutoGet) THEN
			nErrorId := BACnet_ERR_NO_ERROR;
			bDone := FALSE;
		END_IF

	(* READ *)
	1: (* read object property data via ADS *)
		IF TestAndSet(stBACnet_AdsBuffer.bTestSet) THEN
			IF _fbReadProp.bExecute THEN
				IF _fbReadProp.bError THEN
					_i := 100;
					nErrorId := BACnet_ERR_ADS_Read;
					_fbReadProp.bExecute := FALSE;
				ELSIF (NOT _fbReadProp.bBusy) THEN
					_i := 2;
					_fbReadProp.bExecute := FALSE;
					(* prepare pointer *)
					_pSpEventCalEntryDate	:= ADR(stBACnet_AdsBuffer.arrData);
					_pSpEventCalEntryRange	:= ADR(stBACnet_AdsBuffer.arrData);
					_pSpEventCalEntryWnD	:= ADR(stBACnet_AdsBuffer.arrData);
					_pSpEventCalRef			:= ADR(stBACnet_AdsBuffer.arrData);
					(* clear output data *)
					MEMSET(ADR(stExceptSched.arrEntries), 0, SIZEOF(stExceptSched.arrEntries));
					_cbTotalBuf := 0;
					_bNextEvent := TRUE;
				END_IF

			ELSIF (stBACnet_AdsBuffer.iLocked = 0) THEN
				_fbReadProp.bExecute := TRUE;
				(* lock global ADS buffer *)
				stBACnet_AdsBuffer.iLocked := SIZEOF(stBACnet_AdsBuffer.arrData);
			END_IF

			(* release temporary task lock *)
			stBACnet_AdsBuffer.bTestSet := FALSE;
		END_IF

	2: (* select event entry *)
		(* more events? *)
		IF (NOT _bNextEvent) THEN
			(* no more events, exit *)
			_i := 4;
		ELSE
			_i := 3;
			(* check if local buffer is full *)
			IF _iEntry > to_int(BACnet_MaxExSchEntries) THEN
				_i := 4; (* maximum entries reached --> finished *)
			ELSIF ((_pSpEventCalEntryDate^.nEntrySize AND 16#7FFFFFFF) > 0) THEN
				(* initialize first entry *)
				stExceptSched.arrEntries[_iEntry].eEntryType := BACnetCalendarEntryType_None;

				CASE _pSpEventCalEntryDate^.stListEntry.eEventChoice OF

					BACnetSpecialEventChoice_calendarReference:
						_pTimeValue := ADR(_pSpEventCalRef^.stListEntry.stListOfTimeValues);
						stExceptSched.arrEntries[_iEntry].eEntryType := BACnetCalendarEntryType_Ref;
						stExceptSched.arrEntries[_iEntry].stCalRef.tCalObjectId := _pSpEventCalRef^.stListEntry.tCalRef;
						stExceptSched.arrEntries[_iEntry].ePriority := DWORD_TO_INT(_pSpEventCalRef^.stListEntry.iEventPriority);

					BACnetSpecialEventChoice_calendarEntry:
						CASE _pSpEventCalEntryDate^.stListEntry.stCalEntry.eEntryChoice OF
							BACnetCalendarEntryChoice_date:
								_pTimeValue := ADR(_pSpEventCalEntryDate^.stListEntry.stListOfTimeValues);
								stExceptSched.arrEntries[_iEntry].eEntryType := BACnetCalendarEntryType_Date;
								stExceptSched.arrEntries[_iEntry].stDate.stStart := _pSpEventCalEntryDate^.stListEntry.stCalEntry.stDate;
								stExceptSched.arrEntries[_iEntry].stDate.stEnd := _pSpEventCalEntryDate^.stListEntry.stCalEntry.stDate;
								stExceptSched.arrEntries[_iEntry].ePriority := DWORD_TO_INT(_pSpEventCalEntryDate^.stListEntry.iEventPriority);

							BACnetCalendarEntryChoice_dateRange:
								_pTimeValue := ADR(_pSpEventCalEntryRange^.stListEntry.stListOfTimeValues);
								stExceptSched.arrEntries[_iEntry].eEntryType := BACnetCalendarEntryType_DateRange;
								stExceptSched.arrEntries[_iEntry].stDate.stStart := _pSpEventCalEntryRange^.stListEntry.stCalEntry.stStartDate;
								stExceptSched.arrEntries[_iEntry].stDate.stEnd := _pSpEventCalEntryRange^.stListEntry.stCalEntry.stEndDate;
								stExceptSched.arrEntries[_iEntry].ePriority := DWORD_TO_INT(_pSpEventCalEntryRange^.stListEntry.iEventPriority);

							BACnetCalendarEntryChoice_weekNDay:
								_pTimeValue := ADR(_pSpEventCalEntryWnD^.stListEntry.stListOfTimeValues);
								stExceptSched.arrEntries[_iEntry].eEntryType := BACnetCalendarEntryType_WeekNDay;
								stExceptSched.arrEntries[_iEntry].stWeekNDay.iMonth := _pSpEventCalEntryWnD^.stListEntry.stCalEntry.iMonth;
								stExceptSched.arrEntries[_iEntry].stWeekNDay.iWeekOfMonth := _pSpEventCalEntryWnD^.stListEntry.stCalEntry.iWeekOfMonth;
								stExceptSched.arrEntries[_iEntry].stWeekNDay.iDay := _pSpEventCalEntryWnD^.stListEntry.stCalEntry.iDay;
								stExceptSched.arrEntries[_iEntry].ePriority := DWORD_TO_INT(_pSpEventCalEntryWnD^.stListEntry.iEventPriority);

							ELSE
								(* unknown entry choice *)
								nErrorId := BACnet_ERR_UnknownEntryChoice;
								_i := 100;
						END_CASE
					ELSE
						(* unknown event choice *)
						nErrorId := BACnet_ERR_UnknownEventChoice;
						_i := 100;
				END_CASE
			ELSE
				(* mark as invalid *)
				stExceptSched.arrEntries[_iEntry].eEntryType := BACnetCalendarEntryType_None;
			END_IF
		END_IF
		(* reset time value index *)
		_iTv := 0;

	3: (* scan time value list *)
		(* preset next time value flag *)
		_bNextTimeValue := TRUE;
		(* loop till all time values are parsed *)
		WHILE _bNextTimeValue AND _pTimeValue <> 0 DO
			IF ((_pTimeValue^.nEntrySize AND 16#7FFFFFFF) > 0) AND (_iTv <= TO_INT(BACnet_MaxTimeValues)) THEN
				(* time value data available - is it a real type? *)
				IF		_pTimeValue^.stListEntry.stValue.eValueChoice = BACnetDataType_Real
					OR	_pTimeValue^.stListEntry.stValue.eValueChoice = BACnetDataType_Null
				THEN
					(* decide entry type *)
					CASE stExceptSched.arrEntries[_iEntry].eEntryType OF
						BACnetCalendarEntryType_Date,
						BACnetCalendarEntryType_DateRange:
							stExceptSched.arrEntries[_iEntry].arrTimeValue[_iTv].bValid := TRUE;
							stExceptSched.arrEntries[_iEntry].arrTimeValue[_iTv].stTime := _pTimeValue^.stListEntry.stTime;
							stExceptSched.arrEntries[_iEntry].arrTimeValue[_iTv].eType := _pTimeValue^.stListEntry.stValue.eValueChoice;
							IF _pTimeValue^.stListEntry.stValue.cbData = 4 THEN
								MEMCPY(	ADR(stExceptSched.arrEntries[_iEntry].arrTimeValue[_iTv].rValue),
										ADR(_pTimeValue^.stListEntry.stValue.nData),
										SIZEOF(stExceptSched.arrEntries[_iEntry].arrTimeValue[_iTv].rValue)
								);
							ELSE
								stExceptSched.arrEntries[_iEntry].arrTimeValue[_iTv].rValue := F_BACnet_NAN();
							END_IF
							_iTv := _iTv +1;

						BACnetCalendarEntryType_WeekNDay:
							stExceptSched.arrEntries[_iEntry].arrTimeValue[_iTv].bValid := TRUE;
							stExceptSched.arrEntries[_iEntry].arrTimeValue[_iTv].stTime := _pTimeValue^.stListEntry.stTime;
							stExceptSched.arrEntries[_iEntry].arrTimeValue[_iTv].eType := _pTimeValue^.stListEntry.stValue.eValueChoice;
							IF _pTimeValue^.stListEntry.stValue.cbData = 4 THEN
								MEMCPY(	ADR(stExceptSched.arrEntries[_iEntry].arrTimeValue[_iTv].rValue),
										ADR(_pTimeValue^.stListEntry.stValue.nData),
										SIZEOF(stExceptSched.arrEntries[_iEntry].arrTimeValue[_iTv].rValue)
								);
							ELSE
								stExceptSched.arrEntries[_iEntry].arrTimeValue[_iTv].rValue := F_BACnet_NAN();
							END_IF
							_iTv := _iTv +1;

						BACnetCalendarEntryType_Ref:
							stExceptSched.arrEntries[_iEntry].arrTimeValue[_iTv].bValid := TRUE;
							stExceptSched.arrEntries[_iEntry].arrTimeValue[_iTv].stTime := _pTimeValue^.stListEntry.stTime;
							stExceptSched.arrEntries[_iEntry].arrTimeValue[_iTv].eType := _pTimeValue^.stListEntry.stValue.eValueChoice;
							IF _pTimeValue^.stListEntry.stValue.cbData = 4 THEN
								MEMCPY(	ADR(stExceptSched.arrEntries[_iEntry].arrTimeValue[_iTv].rValue),
										ADR(_pTimeValue^.stListEntry.stValue.nData),
										SIZEOF(stExceptSched.arrEntries[_iEntry].arrTimeValue[_iTv].rValue)
								);
							ELSE
								stExceptSched.arrEntries[_iEntry].arrTimeValue[_iTv].rValue := F_BACnet_NAN();
							END_IF
							_iTv := _iTv +1;

					END_CASE

				ELSE
					(* unsupported data type *);
				END_IF

			END_IF

			(* empty entry size or data buffer full, next time value entry *)
			_NextTimeValue();

		END_WHILE

		(* count *)(*
		IF _iTv > 0 THEN
			_iEntry := _iEntry +1;
		END_IF*)
		_iEntry := _iEntry +1;

		(* next event entry *)
		_NextEvent();
		_i := 2;

	4: (* data read and parsed successful *)
		stExceptSched.nGet := stExceptSched.nGet +1;
		_i := 100;

	11: (* lock global ADS buffer *)
		IF TestAndSet(stBACnet_AdsBuffer.bTestSet) THEN
			IF stBACnet_AdsBuffer.iLocked = 0 THEN
				stBACnet_AdsBuffer.iLocked := SIZEOF(stBACnet_AdsBuffer.arrData);
				(* initalize total size counter *)
				_cbTotalBuf := 0;
				(* prepare pointer *)
				_pSpEventCalEntryDate	:= ADR(stBACnet_AdsBuffer.arrData);
				_pSpEventCalEntryRange	:= ADR(stBACnet_AdsBuffer.arrData);
				_pSpEventCalEntryWnD	:= ADR(stBACnet_AdsBuffer.arrData);
				_pSpEventCalRef			:= ADR(stBACnet_AdsBuffer.arrData);
				_pOldEventEntrySize		:= 0;
				(* loop against input data *)
				_i := 12;
			END_IF
			(* release temporary task lock *)
			stBACnet_AdsBuffer.bTestSet := FALSE;
		END_IF

	12: (* write calendar entries date/date range *)
		FOR _iEntry := 0 TO TO_INT(BACnet_MaxExSchEntries) DO

			_pOldTimeValue	:= 0;
			_cbTotalEntry	:= 0;

			IF stExceptSched.arrEntries[_iEntry].eEntryType <> BACnetCalendarEntryType_None THEN
				(* valid entry *)
				CASE stExceptSched.arrEntries[_iEntry].eEntryType OF

					BACnetCalendarEntryType_Date,
					BACnetCalendarEntryType_DateRange:
						(* set special entry choice *)
						IF stExceptSched.arrEntries[_iEntry].eEntryType = BACnetCalendarEntryType_Date THEN
							_pSpEventCalEntryDate^.stListEntry.eEventChoice := BACnetSpecialEventChoice_calendarEntry;
							_pSpEventCalEntryDate^.stListEntry.nRes1 := 0;
							(* set time value pointer *)
							_pTimeValue := ADR(_pSpEventCalEntryDate^.stListEntry.stListOfTimeValues);
						ELSE
							_pSpEventCalEntryRange^.stListEntry.eEventChoice := BACnetSpecialEventChoice_calendarEntry;
							_pSpEventCalEntryRange^.stListEntry.nRes1 := 0;
							(* set time value pointer *)
							_pTimeValue := ADR(_pSpEventCalEntryRange^.stListEntry.stListOfTimeValues);
						END_IF

					BACnetCalendarEntryType_WeekNDay:
						(* set special entry choice *)
						_pSpEventCalEntryWnD^.stListEntry.eEventChoice := BACnetSpecialEventChoice_calendarEntry;
						_pSpEventCalEntryWnD^.stListEntry.nRes1 := 0;
						(* set time value pointer *)
						_pTimeValue := ADR(_pSpEventCalEntryWnD^.stListEntry.stListOfTimeValues);

					BACnetCalendarEntryType_Ref:
						(* set special entry choice *)
						_pSpEventCalRef^.stListEntry.eEventChoice := BACnetSpecialEventChoice_calendarReference;
						_pSpEventCalRef^.stListEntry.nRes1 := 0;
						(* set time value pointer *)
						_pTimeValue := ADR(_pSpEventCalRef^.stListEntry.stListOfTimeValues);

				END_CASE


				(* loop against time values *)
				FOR _iTv := 0 TO to_int(BACnet_MaxTimeValues) DO

					(* valid entry? *)
					IF stExceptSched.arrEntries[_iEntry].arrTimeValue[_iTv].bValid THEN
						(* copy time *)
						_pTimeValue^.stListEntry.stTime := stExceptSched.arrEntries[_iEntry].arrTimeValue[_iTv].stTime;
						_pReal := ADR(_pTimeValue^.stListEntry.stValue.nData);
						_pReal^ := 0.0; (* clear data *)
						(* decide between None and Real type *)
						IF stExceptSched.arrEntries[_iEntry].arrTimeValue[_iTv].eType = BACnetDataType_Real THEN
							(* REAL type *)
							_pTimeValue^.stListEntry.stValue.eValueChoice := BACnetDataType_Real;
							_pTimeValue^.stListEntry.stValue.nRes1 := 0;
							_pTimeValue^.stListEntry.stValue.cbData := SIZEOF(stExceptSched.arrEntries[_iEntry].arrTimeValue[_iTv].rValue);
							MEMCPY(	_pReal,
									ADR(stExceptSched.arrEntries[_iEntry].arrTimeValue[_iTv].rValue),
									MIN(SIZEOF(_pReal^), _pTimeValue^.stListEntry.stValue.cbData)
							);
						ELSE
							(* other or NONE type *)
							_pTimeValue^.stListEntry.stValue.eValueChoice := BACnetDataType_Null;
							_pTimeValue^.stListEntry.stValue.nRes1 := 0;
							_pTimeValue^.stListEntry.stValue.cbData := 0;
						END_IF

						(* calculate time-value entry size *)
						_pTimeValue^.nEntrySize :=	_pTimeValue^.stListEntry.stValue.cbData
												+	SIZEOF(_pTimeValue^.stListEntry.nRes)
												+	SIZEOF(_pTimeValue^.stListEntry.stTime)
												+	SIZEOF(_pTimeValue^.stListEntry.stValue.cbData)
												+	SIZEOF(_pTimeValue^.stListEntry.stValue.eValueChoice)
												+	SIZEOF(_pTimeValue^.stListEntry.stValue.nRes1);

						IF (_iTv > 0 AND _pOldTimeValue <> 0) THEN
							(* next entry flag *)
							_pOldTimeValue^.nEntrySize := _pOldTimeValue^.nEntrySize + 16#80000000;
						END_IF

						(* update time value pointer *)
						_NextTimeValue();

						(* ...and add to total entry size counter *)
						_cbTotalEntry := _cbTotalEntry + _cbTmpSize;

					ELSE
						(* clear entry *)
						_pTimeValue^.nEntrySize := 0;
						_pTimeValue^.stListEntry.stValue.cbData := 0;
					END_IF

				END_FOR

				(* check if time value list is empty *)
				IF _cbTotalEntry = 0 THEN
					(* no time values, set default size *)
					_cbTotalEntry := SIZEOF(_pTimeValue^.nEntrySize) + SIZEOF(_pTimeValue^.nRes);
				END_IF

				(* caclulate event entry size *)
				CASE stExceptSched.arrEntries[_iEntry].eEntryType OF

					BACnetCalendarEntryType_Date:
						(* caclulate event entry size and write into data structure *)
						_pSpEventCalEntryDate^.nEntrySize :=	_cbTotalEntry
															+	SIZEOF(_pSpEventCalEntryDate^.stListEntry.eEventChoice)
															+	SIZEOF(_pSpEventCalEntryDate^.stListEntry.iEventPriority)
															+	SIZEOF(_pSpEventCalEntryDate^.stListEntry.nRes1)
															+	SIZEOF(_pSpEventCalEntryDate^.stListEntry.nRes2)
															+	SIZEOF(_pSpEventCalEntryDate^.stListEntry.nRes3)
															+	SIZEOF(_pSpEventCalEntryDate^.stListEntry.stCalEntry);
						(* copy event data *)
						_pSpEventCalEntryDate^.stListEntry.eEventChoice := BACnetSpecialEventChoice_calendarEntry;
						_pSpEventCalEntryDate^.stListEntry.nRes1 := 0;
						_pSpEventCalEntryDate^.stListEntry.iEventPriority := to_dword(stExceptSched.arrEntries[_iEntry].ePriority);
						_pSpEventCalEntryDate^.stListEntry.stCalEntry.eEntryChoice := BACnetCalendarEntryChoice_date;
						_pSpEventCalEntryDate^.stListEntry.stCalEntry.nRes := 0;
						_pSpEventCalEntryDate^.stListEntry.stCalEntry.stDate := stExceptSched.arrEntries[_iEntry].stDate.stStart;

					BACnetCalendarEntryType_DateRange:
						(* caclulate event entry size and write into data structure *)
						_pSpEventCalEntryRange^.nEntrySize :=	_cbTotalEntry
															+	SIZEOF(_pSpEventCalEntryRange^.stListEntry.eEventChoice)
															+	SIZEOF(_pSpEventCalEntryRange^.stListEntry.iEventPriority)
															+	SIZEOF(_pSpEventCalEntryRange^.stListEntry.nRes1)
															+	SIZEOF(_pSpEventCalEntryRange^.stListEntry.nRes2)
															+	SIZEOF(_pSpEventCalEntryRange^.stListEntry.stCalEntry);
						(* copy event data *)
						_pSpEventCalEntryRange^.stListEntry.eEventChoice := BACnetSpecialEventChoice_calendarEntry;
						_pSpEventCalEntryRange^.stListEntry.nRes1 := 0;
						_pSpEventCalEntryRange^.stListEntry.iEventPriority := to_dword(stExceptSched.arrEntries[_iEntry].ePriority);
						_pSpEventCalEntryRange^.stListEntry.stCalEntry.eEntryChoice := BACnetCalendarEntryChoice_dateRange;
						_pSpEventCalEntryRange^.stListEntry.stCalEntry.nRes := 0;
						_pSpEventCalEntryRange^.stListEntry.stCalEntry.stStartDate := stExceptSched.arrEntries[_iEntry].stDate.stStart;
						_pSpEventCalEntryRange^.stListEntry.stCalEntry.stEndDate := stExceptSched.arrEntries[_iEntry].stDate.stEnd;

					BACnetCalendarEntryType_WeekNDay:
						(* caclulate event entry size and write into data structure *)
						_pSpEventCalEntryWnD^.nEntrySize :=	_cbTotalEntry
															+	SIZEOF(_pSpEventCalEntryWnD^.stListEntry.eEventChoice)
															+	SIZEOF(_pSpEventCalEntryWnD^.stListEntry.iEventPriority)
															+	SIZEOF(_pSpEventCalEntryWnD^.stListEntry.nRes1)
															+	SIZEOF(_pSpEventCalEntryWnD^.stListEntry.nRes2)
															+	SIZEOF(_pSpEventCalEntryWnD^.stListEntry.nRes3)
															+	SIZEOF(_pSpEventCalEntryWnD^.stListEntry.stCalEntry);
						(* copy event data *)
						_pSpEventCalEntryWnD^.stListEntry.eEventChoice := BACnetSpecialEventChoice_calendarEntry;
						_pSpEventCalEntryWnD^.stListEntry.nRes1 := 0;
						_pSpEventCalEntryWnD^.stListEntry.iEventPriority := to_dword(stExceptSched.arrEntries[_iEntry].ePriority);
						_pSpEventCalEntryWnD^.stListEntry.stCalEntry.eEntryChoice := BACnetCalendarEntryChoice_weekNDay;
						_pSpEventCalEntryWnD^.stListEntry.stCalEntry.nRes1 := 0;
						_pSpEventCalEntryWnD^.stListEntry.stCalEntry.iDay := stExceptSched.arrEntries[_iEntry].stWeekNDay.iDay;
						_pSpEventCalEntryWnD^.stListEntry.stCalEntry.iMonth := stExceptSched.arrEntries[_iEntry].stWeekNDay.iMonth;
						_pSpEventCalEntryWnD^.stListEntry.stCalEntry.iWeekOfMonth := stExceptSched.arrEntries[_iEntry].stWeekNDay.iWeekOfMonth;

					BACnetCalendarEntryType_Ref:
						(* caclulate event entry size and write into data structure *)
						_pSpEventCalRef^.nEntrySize :=	_cbTotalEntry
													+	SIZEOF(_pSpEventCalRef^.stListEntry.eEventChoice)
													+	SIZEOF(_pSpEventCalRef^.stListEntry.iEventPriority)
													+	SIZEOF(_pSpEventCalRef^.stListEntry.nRes1)
													+	SIZEOF(_pSpEventCalRef^.stListEntry.nRes2)
													+	SIZEOF(_pSpEventCalRef^.stListEntry.nRes3)
													+	SIZEOF(_pSpEventCalRef^.stListEntry.nRes4)
													+	SIZEOF(_pSpEventCalRef^.stListEntry.tCalRef);
						(* copy event data *)
						_pSpEventCalRef^.stListEntry.eEventChoice := BACnetSpecialEventChoice_calendarReference;
						_pSpEventCalRef^.stListEntry.nRes1 := 0;
						_pSpEventCalRef^.stListEntry.iEventPriority := to_dword(stExceptSched.arrEntries[_iEntry].ePriority);
						_pSpEventCalRef^.stListEntry.tCalRef := stExceptSched.arrEntries[_iEntry].stCalRef.tCalObjectId;

				END_CASE

				(* set next entry flag *)
				IF (_pOldEventEntrySize <> 0) THEN
					_pOldEventEntrySize^ := _pOldEventEntrySize^ + 16#80000000;
				END_IF

				(* next calendar entry *)
				_NextEvent();
			END_IF

		END_FOR

		(* send data *)
		_i := 19;

	19:
		IF _fbWriteProp.bExecute AND (NOT _fbWriteProp.bBusy) THEN
			(* check result *)
			_fbWriteProp.bExecute := FALSE;
			IF _fbWriteProp.bError THEN
				nErrorId := BACnet_ERR_ADS_Write;
			ELSE
				stExceptSched.nSet := stExceptSched.nSet +1;
			END_IF
			_i := 100;
		ELSE
			(* start ADS write *)
			_fbWriteProp.bExecute := TRUE;
		END_IF

	100: (* Done *)
		bDone := (nErrorId = BACnet_ERR_NO_ERROR);
		(* release ADS buffer *)
		stBACnet_AdsBuffer.iLocked := 0;
		(* release data array *)
		stExceptSched.bBusy := FALSE;
		(* go idle *)
		_i := 0;

END_CASE

(* set error flag *)
bError 	:= nErrorId > BACnet_ERR_NO_ERROR;
bBusy 	:= _i > 0;

ACTION _NextEvent:
_bNextEvent := ((_pSpEventCalEntryDate^.nEntrySize AND 16#80000000) = 16#80000000);
_cbTmpSize := _F_BACnet_AlignedSize(_pSpEventCalEntryDate^.nEntrySize AND 16#7FFFFFFF) + SIZEOF(_pSpEventCalEntryDate^.nEntrySize) + SIZEOF(_pSpEventCalEntryDate^.nRes);
_pOldEventEntrySize		:= ADR(_pSpEventCalEntryDate^.nEntrySize);
_pSpEventCalEntryDate	:= _pSpEventCalEntryDate + _cbTmpSize;
_pSpEventCalEntryRange	:= _pSpEventCalEntryRange + _cbTmpSize;
_pSpEventCalEntryWnD	:= _pSpEventCalEntryWnD + _cbTmpSize;
_pSpEventCalRef			:= _pSpEventCalRef + _cbTmpSize;
_cbTotalBuf := _cbTotalBuf + _cbTmpSize;
_pOldTimeValue := 0;
END_ACTION

ACTION _NextTimeValue:
_bNextTimeValue := (_pTimeValue^.nEntrySize AND 16#80000000) = 16#80000000;
_cbTmpSize := 	(_F_BACnet_AlignedSize(_pTimeValue^.nEntrySize) AND 16#7FFFFFFF)
			+	SIZEOF(_pTimeValue^.nEntrySize)
			+	SIZEOF(_pTimeValue^.nRes);
_pOldTimeValue := _pTimeValue;
_pTimeValue := _pTimeValue + _cbTmpSize;
END_ACTION

END_FUNCTION_BLOCK

// POUs/BACnet ADS/Properties/FB_BACnet_LogBufferProperty
FUNCTION_BLOCK FB_BACnet_LogBufferProperty
VAR_INPUT
	tObjectID			: T_BACnet_ObjectIdentifier := 16#FFFFFFFF;
	bAutoGet			: BOOL:=TRUE; (* TRUE = get data from property when ADS connection OR object ID changed *)
	bGet				: BOOL; (* FALSE --> TRUE = get data from property *)
	stStartTime			: ST_BACnet_DateTime := (
							stDate := (nYear := 16#FF, nMonth := 16#FF, nDay := 16#FF),
							stTime := (nHour := 16#FF, nMinute := 16#FF, nSecond := 16#FF, nHundredths := 16#FF)
							); (* Log record beginning from time stStartTime ... (16#FF = unspecified) *)
	stEndTime			: ST_BACnet_DateTime := (
							stDate := (nYear := 16#FF, nMonth := 16#FF, nDay := 16#FF),
							stTime := (nHour := 16#FF, nMinute := 16#FF, nSecond := 16#FF, nHundredths := 16#FF)
							); (* till end time stEndTime (16#FF = unspecified) *)
END_VAR
VAR_IN_OUT
	stAdsConn			: ST_BACnet_AdsConnection;
END_VAR
VAR_OUTPUT
	bDone				: BOOL;
	bBusy				: BOOL;
	bError				: BOOL;
	nErrorId			: UINT;
	stLogBuffer			: ST_BACnet_LogBufferReal;
END_VAR
VAR CONSTANT
	_stMaxTime			: ST_BACnet_Time := (nHour := 23, nMinute := 59, nSecond := 59, nHundredths := 99);
	_stMaxDate			: st_bacnet_date := (nYear := 254, nMonth := 12, nDay := 31, nDayOfWeek := 7);
END_VAR
VAR
	_fbReadProp		: FB_BACnet_ReadProp;
	_fbObjDesc		: FB_BACnet_DescriptionProperty;
	_fbObjName		: FB_BACnet_ObjectNameProperty;
	_i				: INT;
	_rtrigGet		: R_TRIG;

	_pAdsBuf		: POINTER TO BYTE;
	_pLbRecordList	: POINTER TO ST_BACnet_LogRecordList; (* Log buffer - record list *)
	_pLrDatumList	: POINTER TO ST_BACnet_LogDatumList; (* Log record entry - datum list *)

	_iEntry			: INT;

	_bNextRecord	: BOOL;
	_bNextDatum		: BOOL;

	_cbTmpSize		: UDINT;
	_cbTotalBuf		: UDINT;
	_nAdsReloadOld	: USINT;
	_tObjectIDOld	: T_BACnet_ObjectIdentifier := 16#FFFFFFFF;

	_arrRecords		: ARRAY[0..BACnet_MaxLogBufferEntries] OF POINTER TO ST_BACnet_LogRecordList;
	_iNextRecPos	: UDINT;
	_nRecCount		: UDINT;
	_iRec			: UDINT;
	_nMaxSeq		: DWORD; (* max. found sequence no. *)

	_pReal			: POINTER TO REAL;
	_pObjDesc		: POINTER TO STRING;

	_stEndDT		: ST_BACnet_DateTime;
	_nStartTimeDate	: UDINT; (* start time/date since 1900 in 100ms steps *)
	_nEndTimeDate	: UDINT; (* end time/date since 1900 in 100ms steps *)
END_VAR
VAR
	_nTimeStamp		: UDINT;
END_VAR

(*

typedef struct _AnyType
{
      ULONG           nSize;
      BACnetDataTypes dataType;
      //... Data
}AnyType, *PAnyType;

enum BACnetLogRecordChoice
{
      logStatus,              // [0] BACnetLogStatus,
      booleanValue,           // [1] BOOL,
      realValue,              // [2] REAL,
      enumValue,              // [3] ENUMERATED, __ Optionally limited to 32 bits
      unsignedValue,          // [4] Unsigned, __ Optionally limited to 32 bits
      signedValue,            // [5] INTEGER, __ Optionally limited to 32 bits
      bitstringValue,         // [6] BIT STRING, __ Optionally limited to 32 bits
      nullValue,              // [7] NULL,
      failure,                // [8] Error,
      timeChange,             // [9] REAL,
      anyValue,               // [10] ABSTRACT_SYNTAX.&Type __ Optional
};

typedef struct _BACnetLogDatumList
{
      DWORD nEntrySize; // 0x80000000 -> next entry
      DWORD reserved;
      BACnetLogDatum listEntry;
}BACnetLogDatumList, *PBACnetLogDatumList;

typedef struct _BACnetLogDatum
{
      BACnetLogRecordChoice choice;
      union
      {
            DWORD logStatus; // BitString ... of type BACnetLogStatus
            BOOL booleanValue;
            FLOAT realValue;
            EnumerationValueType enumerationValue;
            ULONG unsignedValue;
            DWORD signedValue;
            DWORD bitstringValue;
            DWORD nullValue;
            BACnetError failure; 
            FLOAT timeChange;
            AnyType anyValue; // ABSTRACT-SYNTAX.&Type
      };
}BACnetLogDatum, *PBACnetLogDatum;


typedef struct _BACnetLogRecord
{
      ULONG validFields;
      BACnetDateTime timestamp;          // [0]
      DWORD statusFlags;                       // [2] optional
      BACnetLogDatumList logDatum;  // [1]
}BACnetLogRecord, *PBACnetLogRecord;

typedef struct _BACnetLogRecordList
{
      DWORD nEntrySize; // 0x80000000 -> next entry
      DWORD nSequence;  // "reserved"     -> Number of Sequence begins with 1
      BACnetLogRecord listEntry;
}BACnetLogRecordList, *PBACnetLogRecordList;

*)

(* ADS read *)
_fbReadProp(
	BACnetDevicePort	:= stAdsConn.nAmsPort,
	bExecute			:= ,
	sNetId				:= stAdsConn.sAmsNetId,
	ObjectType			:= F_BACnet_GetObjType(tObjectID),
	PropertyID			:= BACnetPropertyIdentifier_LogBuffer,
	DataType			:= BACnetDataType_LogRecordList,
	ObjectInstance		:= F_BACnet_GetObjInstance(tObjectID),
	ptrValue			:= ADR(stBACnet_AdsBuffer.arrData),
	nLenValue			:= SIZEOF(stBACnet_AdsBuffer.arrData),
	bDone				=> ,
	bBusy				=> ,
	bError				=> ,
	nErrID				=> ,
	nProcessedLen		=> );

_fbObjDesc(
	tObjectID	:= tObjectID,
	bAutoGet	:= FALSE,
	bGet		:= (_i = 1) AND (NOT _fbObjName.bBusy),
	stAdsConn	:= stAdsConn,
	bDone		=> ,
	bBusy		=> ,
	bError		=> ,
	nErrorId	=> ,
	sText		=> );

IF		(_fbObjDesc.bDone AND _fbObjDesc.sText = '')
	OR	_fbObjDesc.bError
THEN
	(* No description found, read name *)
	_fbObjName.bGet := TRUE;
ELSIF _fbObjDesc.bDone THEN
	(* OK, description found *)
	_pObjDesc := ADR(_fbObjDesc.sText);
END_IF

_fbObjName(
	tObjectID	:= tObjectID,
	bAutoGet	:= FALSE,
	bGet		:= ,
	stAdsConn	:= stAdsConn,
	bDone		=> ,
	bBusy		=> ,
	bError		=> ,
	nErrorId	=> ,
	sText		=> );

IF _fbObjName.bDone THEN
	(* OK, name found *)
	_pObjDesc := ADR(_fbObjName.sText);
END_IF
IF (NOT _fbObjName.bBusy) THEN
	_fbObjName.bGet := FALSE;
END_IF

(* trigger start event *)
_rtrigGet(CLK:= bGet, Q=> );

(* state machine *)
CASE _i OF

	0: (* Idle *)
		IF 		_rtrigGet.Q
			OR	(		(		(_nAdsReloadOld <> stAdsConn.nReload)
							OR	(_tObjectIDOld <> tObjectID)
						)
					AND	bAutoGet
				)
		THEN
			IF (NOT stAdsConn.bValid) THEN
				(* ADS connection not valid *)
				nErrorId := BACnet_ERR_INVALID_ADS_CONN;
			ELSIF (NOT stAdsConn.bServer AND NOT stAdsConn.bClient) THEN
				(* not a server nor a client *)
				nErrorId := BACnet_ERR_ADS_NoServerClient;
			ELSE
				_i := 1;
				nErrorId := BACnet_ERR_NO_ERROR;
				(* reset index *)
				_iEntry		:= 0;
				(* remind parameter *)
				_tObjectIDOld := tObjectID;
				_nAdsReloadOld := stAdsConn.nReload;
				(* clear object description index *)
				_pObjDesc := 0;
				(* reset start/end time/date *)
				_nStartTimeDate := 0;
				_nEndTimeDate := 0;
				_stEndDT := stEndTime;
			END_IF
			(* reset done flag *)
			bDone := FALSE;
		END_IF
		IF (NOT bGet) AND (NOT bAutoGet) THEN
			nErrorId := BACnet_ERR_NO_ERROR;
			bDone := FALSE;
		END_IF

	(* READ *)
	1: (* read object property data over ADS *)
		IF TestAndSet(stBACnet_AdsBuffer.bTestSet) THEN
			IF _fbReadProp.bExecute THEN
				IF _fbReadProp.bError THEN
					_i := 100;
					nErrorId := BACnet_ERR_ADS_Read;
					_fbReadProp.bExecute := FALSE;
				ELSIF (NOT _fbReadProp.bBusy) THEN
					_i := 2;
					_fbReadProp.bExecute := FALSE;
					(* prepare pointer *)
					_pAdsBuf := ADR(stBACnet_AdsBuffer.arrData);
					_pLbRecordList := _pAdsBuf;
					(* clear output data *)
					MEMSET(ADR(stLogBuffer.arrEntries), 0, SIZEOF(stLogBuffer.arrEntries));
					stLogBuffer.nCount := 0;
					stLogBuffer.sObjectDesc := '';
					_cbTotalBuf := 0;
					_iNextRecPos := 0;
					_nRecCount := 0;
					_nMaxSeq := 0;
				END_IF

			ELSIF (stBACnet_AdsBuffer.iLocked = 0) THEN
				_fbReadProp.bExecute := TRUE;
				(* lock global ADS buffer *)
				stBACnet_AdsBuffer.iLocked := SIZEOF(stBACnet_AdsBuffer.arrData);
			END_IF

			(* release temporary task lock *)
			stBACnet_AdsBuffer.bTestSet := FALSE;
		END_IF

	2: (* select record list entry *)
		REPEAT (* record list *)

			IF ((_pLbRecordList^.nEntrySize AND 16#7FFFFFFF) > 0) THEN

				(* check sequence order *)
				IF _nMaxSeq > _pLbRecordList^.nSequence THEN
					(* current sequence is lower then previous one - scan entries and sort *)
					FOR _iRec := 0 TO _nRecCount-1 DO
						IF _arrRecords[_iRec]^.nSequence > _pLbRecordList^.nSequence THEN
							(* found higher sequence no. - move *)
							_iNextRecPos := _iRec; (* remind insert position *)
							(* check free space *)
							IF (_nRecCount-1 < BACnet_MaxLogBufferEntries) THEN
								(* enough space at end of list - move *)
								MEMMOVE(	ADR(_arrRecords[_iRec+1]), (* one position up *)
											ADR(_arrRecords[_iRec]), (* free insert position *)
											(_nRecCount - _iRec)*SIZEOF(_arrRecords[0]) (* move all element behind insert position *)
								);
							END_IF
							EXIT; (* leave *)
						END_IF
					END_FOR
				ELSE
					(* remind sequence no. *)
					_nMaxSeq := _pLbRecordList^.nSequence;
				END_IF

				(* insert pointer to record entry *)
				_arrRecords[_iNextRecPos] := _pLbRecordList;
				(* select next free record position and count *)
				_iNextRecPos := _iNextRecPos + 1;
				_nRecCount := _nRecCount + 1;
			END_IF

			(* next record entry *)
			_NextLogRecord();

		UNTIL (		(NOT _bNextRecord) (* no more record entries *)
				OR	(_nRecCount >= (BACnet_MaxLogBufferEntries+1)) (* result buffer full *)
				OR	(_pLbRecordList >= (_pAdsBuf + stBACnet_AdsBuffer.iLocked)) (* ads buffer ending reached *)
			)
		END_REPEAT


		(* preset counter *)
		_iEntry := 0;
		(* scan sorted list *)
		FOR _iRec := 0 TO _nRecCount-1 DO
			(* take first date/time ... *)
			IF (_iRec = 0) THEN
				(* ...and merge with given start time *)
				_nStartTimeDate :=	F_BACnet_Get100msDate(F_BACnet_DateMerge(
										stStartTime.stDate,
										_arrRecords[_iRec]^.listEntry.timestamp.stDate)
									)
								+	F_BACnet_Get100msTime(F_BACnet_TimeMerge(
										stStartTime.stTime,
										_arrRecords[_iRec]^.listEntry.timestamp.stTime)
									);
				(* ...and merge with given end time *)
				IF F_BACnet_TimeUnspecified(_stEndDT.stTime) AND F_BACnet_DateUnspecified(_stEndDT.stDate) THEN
					_stEndDT := _arrRecords[_nRecCount-1]^.listEntry.timestamp;
				ELSE
					(* replace top down all placeholders with start time information *)
					IF _stEndDT.stTime.nHour = 16#FF THEN
						_stEndDT.stTime.nHour := _arrRecords[_iRec]^.listEntry.timestamp.stTime.nHour;
						IF _stEndDT.stTime.nMinute = 16#FF THEN
							_stEndDT.stTime.nMinute := _arrRecords[_iRec]^.listEntry.timestamp.stTime.nMinute;
							IF _stEndDT.stTime.nSecond = 16#FF THEN
								_stEndDT.stTime.nSecond := _arrRecords[_iRec]^.listEntry.timestamp.stTime.nSecond;
								IF _stEndDT.stTime.nHundredths = 16#FF THEN
									_stEndDT.stTime.nHundredths := _arrRecords[_iRec]^.listEntry.timestamp.stTime.nHundredths;
								END_IF
							END_IF
						END_IF
					END_IF
					(* replace time placeholder with maximum time values *)
					_stEndDT.stTime := F_BACnet_TimeMerge(_stEndDT.stTime, _stMaxTime);

					(* replace top down all placeholders with start date information *)
					IF _stEndDT.stDate.nYear = 16#FF THEN
						_stEndDT.stDate.nYear := _arrRecords[_iRec]^.listEntry.timestamp.stDate.nYear;
						IF _stEndDT.stDate.nMonth = 16#FF THEN
							_stEndDT.stDate.nMonth := _arrRecords[_iRec]^.listEntry.timestamp.stDate.nMonth;
							IF _stEndDT.stDate.nDay = 16#FF THEN
								_stEndDT.stDate.nDay := _arrRecords[_iRec]^.listEntry.timestamp.stDate.nDay;
								_stEndDT.stDate.nDayOfWeek := _arrRecords[_iRec]^.listEntry.timestamp.stDate.nDayOfWeek;
							END_IF
						END_IF
					END_IF
					(* replace date placeholder with maximum date values *)
					_stEndDT.stDate := F_BACnet_DateMerge(_stEndDT.stDate, _stMaxDate);
				END_IF

				(* calculate 100ms values for end time/date *)
				_nEndTimeDate := F_BACnet_Get100msTime(_stEndDT.stTime) + F_BACnet_Get100msDate(_stEndDT.stDate);
				IF _nEndTimeDate <= (		F_BACnet_Get100msTime(_arrRecords[_iRec]^.listEntry.timestamp.stTime)
										+	F_BACnet_Get100msDate(_arrRecords[_iRec]^.listEntry.timestamp.stDate)
									)
				THEN
					(* end time is lower than start time - set maximum value *)
					_nEndTimeDate := 	16#FFFFFFFF;
				END_IF
			END_IF

			(* initialize datum list pointer *)
			_pLrDatumList := ADR(_arrRecords[_iRec]^.listEntry.logDatum);

			REPEAT (* datum list *)

				(* check if local buffer is full *)
				IF _iEntry > to_int(BACnet_MaxLogBufferEntries) THEN
					(* maximum entries reached --> finished *)
					_i := 4;
				ELSIF (_pLrDatumList^.nEntrySize AND 16#7FFFFFFF) > 0 THEN
					(* check time range *)
					_nTimeStamp :=	F_BACnet_Get100msDate(_arrRecords[_iRec]^.listEntry.timestamp.stDate)
								+	F_BACnet_Get100msTime(_arrRecords[_iRec]^.listEntry.timestamp.stTime);
					IF		(_nTimeStamp >= _nStartTimeDate) AND (_nTimeStamp <= _nEndTimeDate)
						AND	(_pLrDatumList^.listEntry.choice = BACnetLogRecordChoice_realValue)
					THEN
						(* append entry *)
						stLogBuffer.arrEntries[_iEntry].stDateTime := _arrRecords[_iRec]^.listEntry.timestamp;
						stLogBuffer.arrEntries[_iEntry].nTimeStamp := _nTimeStamp;
						_pReal := ADR(_pLrDatumList^.listEntry.nData);
						stLogBuffer.arrEntries[_iEntry].fValue := _pReal^;
						(* count up *)
						_iEntry := _iEntry + 1;
					END_IF
				END_IF

				(* next datum entry *)
				_NextLogDatum();

			UNTIL	(NOT _bNextDatum)
				OR	(_i <> 2)
			END_REPEAT

			(* exit if state changed *)
			IF _i <> 2 THEN EXIT; END_IF
		END_FOR
		_i := 4;


	4: (* wait on object description *)
		IF (NOT _fbObjDesc.bBusy) AND (NOT _fbObjName.bBusy) THEN
			(* set description *)
			IF _pObjDesc <> 0 THEN
				stLogBuffer.sObjectDesc := _pObjDesc^;
			ELSE
				stLogBuffer.sObjectDesc := F_BACnet_GetObjectIdString(tObjectID);
			END_IF
			(* set count *)
			stLogBuffer.nCount := TO_UDINT(_iEntry);
			stLogBuffer.nGet := stLogBuffer.nGet + 1;
			_i := 100;
		END_IF

	100: (* Done *)
		bDone := (nErrorId = BACnet_ERR_NO_ERROR);
		(* release ADS buffer *)
		stBACnet_AdsBuffer.iLocked := 0;
		(* go idle *)
		_i := 0;

END_CASE

(* set error flag *)
bError 	:= nErrorId > BACnet_ERR_NO_ERROR;
bBusy 	:= _i > 0;

ACTION _NextLogDatum:
_bNextDatum := (_pLrDatumList^.nEntrySize AND 16#80000000) = 16#80000000;
_cbTmpSize := 	(_F_BACnet_AlignedSize(_pLrDatumList^.nEntrySize) AND 16#7FFFFFFF)
			+	SIZEOF(_pLrDatumList^.nEntrySize)
			+	SIZEOF(_pLrDatumList^.reserved);
_pLrDatumList := _pLrDatumList + _cbTmpSize;
END_ACTION

ACTION _NextLogRecord:
_bNextRecord := ((_pLbRecordList^.nEntrySize AND 16#80000000) = 16#80000000);
_cbTmpSize := _F_BACnet_AlignedSize(_pLbRecordList^.nEntrySize AND 16#7FFFFFFF) + SIZEOF(_pLbRecordList^.nEntrySize) + SIZEOF(_pLbRecordList^.nSequence);
_pLbRecordList	:= _pLbRecordList + _cbTmpSize;
_cbTotalBuf := _cbTotalBuf + _cbTmpSize;
END_ACTION

END_FUNCTION_BLOCK

// POUs/BACnet Helper/DateTime/F_BACnet_Get100msDate
FUNCTION F_BACnet_Get100msDate : UDINT (* Returns date as 100ms value from 1900 (if year and month are specified!) *)
VAR_INPUT
	stBACnetDate		: ST_BACnet_Date;
END_VAR
VAR
	iValue : UDINT;
	i : BYTE;
	stDate : ST_BACnet_Date;
END_VAR

iValue := 0;
IF stBACnetDate.nYear < 16#FF THEN
	iValue := iValue + BYTE_TO_UDINT(stBACnetDate.nYear) * 365 * 24 * 60 * 60 * 10;
	IF stBACnetDate.nDay >= 1 AND stBACnetDate.nDay <= 12 THEN
		stDate := stBACnetDate;
		FOR i := 1 TO stBACnetDate.nMonth-1 DO
			stDate.nMonth := i;
			iValue := iValue + F_BACnet_DaysInMonth(stDate) * 24 * 60 * 60 * 10;
		END_FOR
	END_IF
END_IF
IF stBACnetDate.nDay >= 1 AND stBACnetDate.nDay <= 31 THEN
	iValue := iValue + BYTE_TO_UDINT(stBACnetDate.nDay) * 24 * 60 * 60 * 10;
END_IF
F_BACnet_Get100msDate := iValue;

END_FUNCTION

// POUs/BACnet Helper/DateTime/F_BACnet_DaysInMonth
FUNCTION F_BACnet_DaysInMonth : UDINT (* Returns the numbers of days in given month - 16#FFFFFFFF = unspecified *)
VAR_INPUT
	stBACnetDate		: ST_BACnet_Date;
END_VAR
VAR
	isLeapYear			: BOOL;
	nYear				: UDINT;
END_VAR

IF (stBACnetDate.nMonth = 16#FF) OR (stBACnetDate.nYear = 16#FF) THEN
	(* month and/or year is unspecified *)
	F_BACnet_DaysInMonth := 16#FFFFFFFF;
ELSIF	stBACnetDate.nMonth = 1
	OR	stBACnetDate.nMonth = 3
	OR	stBACnetDate.nMonth = 5
	OR	stBACnetDate.nMonth = 7
	OR	stBACnetDate.nMonth = 8
	OR	stBACnetDate.nMonth = 10
	OR	stBACnetDate.nMonth = 12
THEN
	F_BACnet_DaysInMonth := 31;
ELSE
	IF (stBACnetDate.nMonth = 2) THEN
		(* calculate absolute your number *)
		nYear := stBACnetDate.nYear + 1900;
		(* and check if it is a leap year *)
		isLeapYear := (nYear MOD 4 = 0) AND ((nYear MOD 100 <> 0) OR (nYear MOD 400 = 0));
		(* decide february amount of days *)
		IF (isLeapYear) THEN
		  F_BACnet_DaysInMonth := 29;
		ELSE
		  F_BACnet_DaysInMonth := 28;
		END_IF
	ELSE
		F_BACnet_DaysInMonth := 30;
	END_IF
END_IF

END_FUNCTION

// POUs/BACnet Helper/DateTime/F_BACnet_DateMerge
FUNCTION F_BACnet_DateMerge : ST_BACnet_Date (* This function replacing placeholders in both dates and returning the result (if no placeholder is given, date1 will be prefered) *)
VAR_INPUT
	stDate1		: ST_BACnet_Date;
	stDate2		: ST_BACnet_Date;
END_VAR
VAR
END_VAR

IF stDate1.nDay = 16#FF THEN
	F_BACnet_DateMerge.nDay := F_BACnet_CheckDay(stDate2.nDay);
ELSE
	F_BACnet_DateMerge.nDay := F_BACnet_CheckDay(stDate1.nDay);
END_IF
IF stDate1.nDayOfWeek = 16#FF THEN
	F_BACnet_DateMerge.nDayOfWeek := F_BACnet_CheckDayOfWeek(stDate2.nDayOfWeek);
ELSE
	F_BACnet_DateMerge.nDayOfWeek := F_BACnet_CheckDayOfWeek(stDate1.nDayOfWeek);
END_IF
IF stDate1.nMonth = 16#FF THEN
	F_BACnet_DateMerge.nMonth := F_BACnet_CheckMonth(stDate2.nMonth);
ELSE
	F_BACnet_DateMerge.nMonth := F_BACnet_CheckMonth(stDate1.nMonth);
END_IF
IF stDate1.nYear = 16#FF THEN
	F_BACnet_DateMerge.nYear := F_BACnet_CheckYear(stDate2.nYear);
ELSE
	F_BACnet_DateMerge.nYear := F_BACnet_CheckYear(stDate1.nYear);
END_IF

END_FUNCTION

// POUs/BACnet Helper/DateTime/F_BACnet_CheckDay
FUNCTION F_BACnet_CheckDay : USINT

VAR
END_VAR
(*All VAR_IN_OUT variables have been moved to the end of the declaration due to compatibility reasons*)
VAR_IN_OUT
	nIn	: BYTE;
END_VAR

IF nIn > 32 OR nIn = 0 THEN
	F_BACnet_CheckDay := 255;
ELSE
	F_BACnet_CheckDay := nIn;
END_IF
nIn := F_BACnet_CheckDay;

END_FUNCTION

// POUs/BACnet Helper/DateTime/F_BACnet_CheckDayOfWeek
FUNCTION F_BACnet_CheckDayOfWeek : USINT

VAR
END_VAR
(*All VAR_IN_OUT variables have been moved to the end of the declaration due to compatibility reasons*)
VAR_IN_OUT
	nIn	: BYTE;
END_VAR

IF nIn > 7 OR nIn = 0 THEN
	F_BACnet_CheckDayOfWeek := 255;
ELSE
	F_BACnet_CheckDayOfWeek := nIn;
END_IF
nIn := F_BACnet_CheckDayOfWeek;

END_FUNCTION

// POUs/BACnet Helper/DateTime/F_BACnet_CheckMonth
FUNCTION F_BACnet_CheckMonth : USINT

VAR
END_VAR
(*All VAR_IN_OUT variables have been moved to the end of the declaration due to compatibility reasons*)
VAR_IN_OUT
	nIn	: BYTE;
END_VAR

IF nIn > 14 OR nIn = 0 THEN
	F_BACnet_CheckMonth := 255;
ELSE
	F_BACnet_CheckMonth := nIn;
END_IF
nIn := F_BACnet_CheckMonth;

END_FUNCTION

// POUs/BACnet Helper/DateTime/F_BACnet_CheckYear
FUNCTION F_BACnet_CheckYear : USINT

VAR
END_VAR
(*All VAR_IN_OUT variables have been moved to the end of the declaration due to compatibility reasons*)
VAR_IN_OUT
	nIn	: BYTE;
END_VAR

F_BACnet_CheckYear := nIn;
nIn := F_BACnet_CheckYear;

END_FUNCTION

// POUs/BACnet Helper/DateTime/F_BACnet_Get100msTime
FUNCTION F_BACnet_Get100msTime : UDINT (* Returns time as 100ms value from 00:00:00.0 *)
VAR_INPUT
	stBACnetTime : ST_BACnet_Time;
END_VAR
VAR
	iValue		: UDINT;
END_VAR

iValue := 0;
IF (stBACnetTime.nHour < 16#FF) THEN
	iValue := iValue + BYTE_TO_UDINT(stBACnetTime.nHour) * 60 * 60 * 10;
END_IF
IF (stBACnetTime.nMinute < 16#FF) THEN
	iValue := iValue + BYTE_TO_UDINT(stBACnetTime.nMinute) * 60 * 10;
END_IF
IF (stBACnetTime.nSecond < 16#FF) THEN
	iValue := iValue + BYTE_TO_UDINT(stBACnetTime.nSecond) * 10;
END_IF
IF (stBACnetTime.nHundredths < 16#FF) THEN
	iValue := iValue + BYTE_TO_UDINT(stBACnetTime.nHundredths) / 10;
END_IF
F_BACnet_Get100msTime := iValue;

END_FUNCTION

// POUs/BACnet Helper/DateTime/F_BACnet_TimeMerge
FUNCTION F_BACnet_TimeMerge : ST_BACnet_Time (* This function replaces placeholder in time1 with time2 and returning the result (if no placeholder is given, time1 will be prefered) *)
VAR_INPUT
	stTime1		: ST_BACnet_Time;
	stTime2		: ST_BACnet_Time;
END_VAR
VAR
END_VAR

IF stTime1.nHour = 16#FF THEN
	F_BACnet_TimeMerge.nHour := F_BACnet_CheckHour(stTime2.nHour);
ELSE
	F_BACnet_TimeMerge.nHour := F_BACnet_CheckHour(stTime1.nHour);
END_IF
IF stTime1.nHundredths = 16#FF THEN
	F_BACnet_TimeMerge.nHundredths := F_BACnet_CheckHundredths(stTime2.nHundredths);
ELSE
	F_BACnet_TimeMerge.nHundredths := F_BACnet_CheckHundredths(stTime1.nHundredths);
END_IF
IF stTime1.nMinute = 16#FF THEN
	F_BACnet_TimeMerge.nMinute := F_BACnet_CheckMinute(stTime2.nMinute);
ELSE
	F_BACnet_TimeMerge.nMinute := F_BACnet_CheckMinute(stTime1.nMinute);
END_IF
IF stTime1.nSecond = 16#FF THEN
	F_BACnet_TimeMerge.nSecond := F_BACnet_CheckSecond(stTime2.nSecond);
ELSE
	F_BACnet_TimeMerge.nSecond := F_BACnet_CheckSecond(stTime1.nSecond);
END_IF

END_FUNCTION

// POUs/BACnet Helper/DateTime/F_BACnet_CheckHour
FUNCTION F_BACnet_CheckHour : USINT

VAR
END_VAR
(*All VAR_IN_OUT variables have been moved to the end of the declaration due to compatibility reasons*)
VAR_IN_OUT
	nIn	: BYTE;
END_VAR

IF nIn > 23 THEN
	F_BACnet_CheckHour := 255;
ELSE
	F_BACnet_CheckHour := nIn;
END_IF
nIn := F_BACnet_CheckHour;

END_FUNCTION

// POUs/BACnet Helper/DateTime/F_BACnet_CheckHundredths
FUNCTION F_BACnet_CheckHundredths : USINT

VAR
END_VAR
(*All VAR_IN_OUT variables have been moved to the end of the declaration due to compatibility reasons*)
VAR_IN_OUT
	nIn	: BYTE;
END_VAR

IF nIn > 99 THEN
	F_BACnet_CheckHundredths := 255;
ELSE
	F_BACnet_CheckHundredths := nIn;
END_IF
nIn := F_BACnet_CheckHundredths;

END_FUNCTION

// POUs/BACnet Helper/DateTime/F_BACnet_CheckMinute
FUNCTION F_BACnet_CheckMinute : USINT

VAR
END_VAR
(*All VAR_IN_OUT variables have been moved to the end of the declaration due to compatibility reasons*)
VAR_IN_OUT
	nIn	: BYTE;
END_VAR

IF nIn > 59 THEN
	F_BACnet_CheckMinute := 255;
ELSE
	F_BACnet_CheckMinute := nIn;
END_IF
nIn := F_BACnet_CheckMinute;

END_FUNCTION

// POUs/BACnet Helper/DateTime/F_BACnet_CheckSecond
FUNCTION F_BACnet_CheckSecond : USINT

VAR
END_VAR
(*All VAR_IN_OUT variables have been moved to the end of the declaration due to compatibility reasons*)
VAR_IN_OUT
	nIn	: BYTE;
END_VAR

IF nIn > 59 THEN
	F_BACnet_CheckSecond := 255;
ELSE
	F_BACnet_CheckSecond := nIn;
END_IF
nIn := F_BACnet_CheckSecond;

END_FUNCTION

// POUs/BACnet Helper/DateTime/F_BACnet_TimeUnspecified
FUNCTION F_BACnet_TimeUnspecified : BOOL
VAR_INPUT
	stTime		: ST_BACnet_Time;
END_VAR

F_BACnet_TimeUnspecified := (stTime.nHour = 16#FF) AND (stTime.nHundredths = 16#FF) AND (stTime.nMinute = 16#FF) AND (stTime.nSecond = 16#FF);

END_FUNCTION

// POUs/BACnet Helper/DateTime/F_BACnet_DateUnspecified
FUNCTION F_BACnet_DateUnspecified : BOOL
VAR_INPUT
	stDate		: ST_BACnet_Date;
END_VAR

F_BACnet_DateUnspecified := (stDate.nDay = 16#FF) AND (stDate.nDayOfWeek = 16#FF) AND (stDate.nMonth = 16#FF) AND (stDate.nYear = 16#FF);

END_FUNCTION

// POUs/BACnet Helper/String/F_BACnet_GetObjectIdString
FUNCTION F_BACnet_GetObjectIdString : STRING
VAR_INPUT
	tObjectID : T_BACnet_ObjectIdentifier := 16#FFFFFFFF;
END_VAR
VAR
	nObjType	: DINT;
	nObjInstance: UDINT;
END_VAR

nObjType	:= F_BACnet_GetObjType(tObjectID);
nObjInstance:= F_BACnet_GetObjInstance(tObjectID);
IF nObjType >= 0 AND nObjType < BACnetObjectType_ZCount THEN
	F_BACnet_GetObjectIdString := CONCAT(CONCAT(arrBACnet_ObjectTypeNameShort[nObjType], ':'), UDINT_TO_STRING(nObjInstance));
ELSE
	F_BACnet_GetObjectIdString := CONCAT('???:', UDINT_TO_STRING(nObjInstance));
END_IF

END_FUNCTION

// POUs/BACnet ADS/Properties/FB_BACnet_ObjectNameProperty
FUNCTION_BLOCK FB_BACnet_ObjectNameProperty
VAR_INPUT
	tObjectID			: T_BACnet_ObjectIdentifier := 16#FFFFFFFF;
	bAutoGet			: BOOL:=TRUE; (* TRUE = get data from property when ADS connection OR object ID changed *)
	bGet				: BOOL; (* FALSE --> TRUE = get data from property *)
END_VAR
VAR_IN_OUT
	stAdsConn			: ST_BACnet_AdsConnection;
END_VAR
VAR_OUTPUT
	bDone				: BOOL;
	bBusy				: BOOL;
	bError				: BOOL;
	nErrorId			: UINT;
	sText				: T_MaxString; (* Object name *)
END_VAR
VAR
	_fbReadProp		: FB_BACnet_ReadProp;
	_i				: INT;
	_rtrigGetSet	: R_TRIG;
	_nAdsReloadOld	: USINT;
	_tObjectIDOld	: T_BACnet_ObjectIdentifier := 16#FFFFFFFF;
	_StringExtDecode: FB_BACnet_StringExtDecode;
END_VAR


(* ADS read *)
_fbReadProp(
	BACnetDevicePort	:= stAdsConn.nAmsPort,
	bExecute			:= ,
	sNetId				:= stAdsConn.sAmsNetId,
	ObjectType			:= F_BACnet_GetObjType(tObjectID),
	PropertyID			:= BACnetPropertyIdentifier_ObjectName,
	DataType			:= BACnetDataType_CharacterStringExt,
	ObjectInstance		:= F_BACnet_GetObjInstance(tObjectID),
	ptrValue			:= ADR(sText),
	nLenValue			:= SIZEOF(sText)-1,
	bDone				=> ,
	bBusy				=> ,
	bError				=> ,
	nErrID				=> ,
	nProcessedLen		=> );

(* trigger start event *)
_rtrigGetSet(CLK:= bGet, Q=> );

(* state machine *)
CASE _i OF

	0: (* Idle *)
		IF		(		(		_rtrigGetSet.Q
							OR	(_nAdsReloadOld <> stAdsConn.nReload)
							OR	(_tObjectIDOld <> tObjectID)
						)
					AND	bAutoGet
				)
			OR	_rtrigGetSet.Q
		THEN
			IF (NOT stAdsConn.bValid) THEN
				(* ADS connection not valid *)
				nErrorId := BACnet_ERR_INVALID_ADS_CONN;
			ELSIF (NOT stAdsConn.bServer AND NOT stAdsConn.bClient) THEN
				(* not a server nor a client *)
				nErrorId := BACnet_ERR_ADS_NoServerClient;
			ELSE
				nErrorId := BACnet_ERR_NO_ERROR;
				_i := 1;
				sText := '';
				(* remind ADS reload counter and parameter *)
				_nAdsReloadOld := stAdsConn.nReload;
				_tObjectIDOld := tObjectID;
			END_IF
			(* reset done flag *)
			bDone := FALSE;
		END_IF
		IF (NOT bGet) AND (NOT bAutoGet) THEN
			nErrorId := BACnet_ERR_NO_ERROR;
			bDone := FALSE;
		END_IF

	(* READ *)
	1: (* read object property data over ADS *)
		IF _fbReadProp.bExecute THEN
			IF _fbReadProp.bError THEN
				_i := 100;
				nErrorId := BACnet_ERR_ADS_Read;
				_fbReadProp.bExecute := FALSE;
			ELSIF (NOT _fbReadProp.bBusy) THEN
				_fbReadProp.bExecute := FALSE;
				(* decode property data *)
				_StringExtDecode(
					pChrStringExt	:= ADR(sText),
					cbOutSize		:= _fbReadProp.nProcessedLen,
					pOutString		:= ADR(sText),
					bValid			=> ,
					bOverflow		=> ,
					nLength			=> ,
					eSrcEncoding	=> );
				(* check overflow flag *)
				IF _StringExtDecode.bOverflow THEN
					nErrorId := BACnet_ERR_ADS_BufferSize;
				END_IF
				(* DONE *)
				_i := 100;
			END_IF
		ELSE
			_fbReadProp.bExecute := TRUE;
		END_IF

	100: (* Done *)
		bDone := (nErrorId = BACnet_ERR_NO_ERROR);
		_i := 0;

END_CASE

(* set error flag *)
bError 	:= nErrorId > BACnet_ERR_NO_ERROR;
bBusy 	:= _i > 0;

END_FUNCTION_BLOCK

// POUs/BACnet ADS/Properties/FB_BACnet_ObjectListProperty
FUNCTION_BLOCK FB_BACnet_ObjectListProperty
VAR_INPUT
	bAutoGet			: BOOL:=TRUE; (* TRUE = get data from property when ADS connection OR object ID changed *)
	bGet				: BOOL; (* FALSE --> TRUE = get data from property *)
	bTypeFilter			: BOOL; (* activate input "eObjectTypeFilter" *)
	eObjType			: E_BACnetObjectType; (* select the object type that is scanned *)
END_VAR
VAR_IN_OUT
	stAdsConn			: ST_BACnet_AdsConnection;
END_VAR
VAR_OUTPUT
	bDone				: BOOL;
	bBusy				: BOOL;
	bError				: BOOL;
	nErrorId			: UINT;
	stObjIDList			: ST_BACnet_ObjectIdentifierList;
END_VAR
VAR
	_fbReadProp			: FB_BACnet_ReadProp;
	_i					: INT;
	_cbPropSize			: UDINT;
	_cbMemCpy			: UDINT;
	_nEntryCount		: UDINT;
	_iScan				: UDINT;
	_pEntry				: POINTER TO T_BACnet_ObjectIdentifier;
	_cbAdsBuf			: UDINT;
	_rtrigGetSet		: R_TRIG;
	_nAdsReloadOld		: USINT;
	_bUseObjTypeFilterOld: BOOL;
	_eObjTypeFilterOld	: E_BACnetObjectType;
	_nDeviceIdOld		: DWORD := 16#FFFFFFFF;
END_VAR

(* ADS read *);
_fbReadProp(
	BACnetDevicePort	:= stAdsConn.nAmsPort,
	bExecute			:= ,
	ObjectInstance		:= F_BACnet_GetObjInstance(stAdsConn.nDeviceId),
	ObjectType			:= BACnetObjectType_Device,
	sNetId				:= stAdsConn.sAmsNetId,
	PropertyID			:= BACnetPropertyIdentifier_ObjectList,
	DataType			:= BACnetDataType_ObjectIdentifierArr,
	ptrValue			:= ADR(stBACnet_AdsBuffer.arrData),
	nLenValue			:= SIZEOF(stBACnet_AdsBuffer.arrData),
	bDone				=> ,
	bBusy				=> ,
	bError				=> ,
	nErrID				=> ,
	nProcessedLen		=> );

(* trigger start event *)
_rtrigGetSet(CLK:= bGet, Q=> );

(* state machine *)
CASE _i OF

	0: (* Idle *)
		IF		(		(
								(_nAdsReloadOld <> stAdsConn.nReload)
							OR	(_bUseObjTypeFilterOld <> bTypeFilter)
							OR	((_eObjTypeFilterOld <> eObjType) AND bTypeFilter)
							OR	(_nDeviceIdOld <> stAdsConn.nDeviceId)
						)
					AND	bAutoGet
				)
			OR	_rtrigGetSet.Q
		THEN
			IF (NOT stAdsConn.bValid) THEN
				(* ADS connection not valid *)
				nErrorId := BACnet_ERR_INVALID_ADS_CONN;
			ELSIF (NOT stAdsConn.bServer AND NOT stAdsConn.bClient) THEN
				(* not a server nor a client *)
				nErrorId := BACnet_ERR_ADS_NoServerClient;
			ELSE
				nErrorId := BACnet_ERR_NO_ERROR;
				_i := 1;
				(* remind ADS reload counter and parameter *)
				_nAdsReloadOld := stAdsConn.nReload;
				_bUseObjTypeFilterOld := bTypeFilter;
				_eObjTypeFilterOld := eObjType;
				_nDeviceIdOld := stAdsConn.nDeviceId;
			END_IF
			(* reset done flag *)
			bDone := FALSE;
		END_IF
		IF (NOT bGet) AND (NOT bAutoGet) THEN
			nErrorId := BACnet_ERR_NO_ERROR;
			bDone := FALSE;
		END_IF

	(* READ *)
	1: (* read object property data via ADS *)
		IF TestAndSet(stBACnet_AdsBuffer.bTestSet) THEN
			IF _fbReadProp.bExecute THEN
				IF _fbReadProp.bError THEN
					_i := 100;
					nErrorId := BACnet_ERR_ADS_Read;
					_fbReadProp.bExecute := FALSE;
				ELSIF (NOT _fbReadProp.bBusy) THEN
					_fbReadProp.bExecute := FALSE;
					_cbPropSize := _fbReadProp.nProcessedLen;
					(* clear output data *)
					MEMSET(ADR(stObjIDList), 0, SIZEOF(stObjIDList));
					(* check if the ADS buffer reached its ending *)
					IF _cbPropSize > _cbAdsBuf THEN
						(* ADS buffer too small *)
						nErrorId := BACnet_ERR_ADS_BufferSize;
						(* reduce size of data to copy *)
						IF (_cbAdsBuf MOD 4) <> 0 THEN
							_cbPropSize := _F_BACnet_AlignedSize(_cbAdsBuf - 4);
						ELSE
							_cbPropSize := _cbAdsBuf;
						END_IF
					END_IF

					(* filter object type or not? *)
					IF NOT bTypeFilter THEN
						(* copy all from ADS buffer *)
						_cbMemCpy := MEMCPY(	ADR(stObjIDList.arrObjList),
												ADR(stBACnet_AdsBuffer.arrData),
												MIN(_cbPropSize, SIZEOF(stObjIDList.arrObjList))
						);
						IF _cbMemCpy < _cbPropSize THEN
							(* not all property data copied *)
							nErrorId := BACnet_ERR_ADS_TooManyObjects;
						END_IF
						(* how many entries read? *)
						stObjIDList.nEntries := _cbMemCpy / 4;
					ELSE
						(* filter - scan entry by entry *)
						_nEntryCount := _cbPropSize / 4;
						_iScan := 0;
						_pEntry := ADR(stBACnet_AdsBuffer.arrData);
						_cbPropSize := TO_UDINT(_pEntry) + _cbPropSize;
						(* scan entry by entry and add to list if matching with filter *)
						WHILE (		(TO_UDINT(_pEntry) + 4) <= _cbPropSize)
								AND	(_iScan < _nEntryCount)
						DO
							IF F_BACnet_GetObjType(_pEntry^) = eObjType THEN
								(* add item to list *)
								stObjIDList.arrObjList[stObjIDList.nEntries] := _pEntry^;
								stObjIDList.nEntries := stObjIDList.nEntries + 1;
							END_IF
							(* count up *)
							_iScan := _iScan + 1;
							_pEntry := _pEntry + SIZEOF(_pEntry^);
						END_WHILE
					END_IF
					(* DONE *)
					_i := 100;
				END_IF

			ELSIF (stBACnet_AdsBuffer.iLocked = 0) THEN
				_fbReadProp.bExecute := TRUE;
				(* lock global ADS buffer *)
				_cbAdsBuf := SIZEOF(stBACnet_AdsBuffer.arrData);
				stBACnet_AdsBuffer.iLocked := TO_DINT(_cbAdsBuf);
			END_IF

			(* release temporary task lock *)
			stBACnet_AdsBuffer.bTestSet := FALSE;
		END_IF

	100: (* Done *)
		bDone := (nErrorId = BACnet_ERR_NO_ERROR);
		(* release ADS buffer *)
		stBACnet_AdsBuffer.iLocked := 0;
		_i := 0;

END_CASE

(* set error flag *)
bError 	:= nErrorId > BACnet_ERR_NO_ERROR;
bBusy 	:= _i > 0;

END_FUNCTION_BLOCK

// POUs/BACnet ADS/Properties/FB_BACnet_RecipientListProperty
FUNCTION_BLOCK FB_BACnet_RecipientListProperty
VAR_INPUT
	tObjectID			: T_BACnet_ObjectIdentifier := 16#FFFFFFFF;
	bAutoGet			: BOOL:=TRUE; (* TRUE = get data from property when ADS connection OR object ID changed *)
	bGet				: BOOL; (* FALSE --> TRUE = get data from property *)
	bSet				: BOOL; (* FALSE --> TRUE = set data into property *)
END_VAR
VAR_IN_OUT
	stAdsConn			: ST_BACnet_AdsConnection;
	stRecipients		: ST_BACnet_RecipientListDevice;
END_VAR
VAR_OUTPUT
	bDone				: BOOL;
	bBusy				: BOOL;
	bError				: BOOL;
	nErrorId			: UINT;
END_VAR
VAR
	_fbReadProp		: FB_BACnet_ReadProp;
	_fbWriteProp	: FB_BACnet_WriteProp;
	_i				: INT;
	_rtrigGet		: R_TRIG;
	_rtrigSet		: R_TRIG;

	_nAdsReloadOld	: USINT;
	_tObjectIDOld	: T_BACnet_ObjectIdentifier := 16#FFFFFFFF;

	_iEntryCheck	: UDINT;
	_iEntry			: INT;
	_iDataEntry		: INT;
	_iReadElems		: UDINT;

	_pEntryList		: POINTER TO T_BACnet_DestinationDeviceArray;

	_cbDestList		: UDINT;
	_cbDestListElem	: UDINT;
END_VAR

(*
	enum BACnetRecipient_Choice
	{
	      device,
	      address
	};
	
	typedef struct _BACnetObjectIdentifier
	{
	      union
	      {
	            struct 
	            {
	                  DWORD objInst : 22;
	                  DWORD objType : 10;
	            };
	            DWORD objId;
	      };
	}BACnetObjectIdentifier, *PBACnetObjectIdentifier;
	
	typedef struct _BACnetAddress
	{
	      BACnetAddressChoice choice;
	      BYTE layerAddress[7]; // MS/TP...LonTalk 
	      BYTE reserved;
	      USHORT      network_number;
	}BACnetAddress, *PBACnetAddress;
	
	enum BACnetAddressChoice
	{
	      Ethernet,
	      Arcnet,
	      MsTp,
	      LonTalk,
	      LonTalkNeuronId,
	      Address_3,
	      Address_4,
	      Address_5,
	      Broadcast
	};
	
	typedef struct _BACnetRecipient
	{ 
	      BACnetRecipient_Choice choiceField;
	      union
	      {
	            BACnetObjectIdentifier  device;
	            BACnetAddress           address;
	      };
	}BACnetRecipient,*PBACnetRecipient;
		
	typedef struct _BACnetDestination
	{ 
	      ULONG                              validDays;  //Bitfield of BACnetDaysOfWeek
	      BACnetTime                         fromTime;
	      BACnetTime                         toTime;
	      BACnetRecipient                    recipient;
	      ULONG                              processIdentifier;
	      DWORD                              transitionsBits;  // BACnetEventTransitionBits
	      BOOL                               issueConfirmedNotifications;
	}BACnetDestination,*PBACnetDestination;


*)

(* ADS read *)
_fbReadProp(
	BACnetDevicePort	:= stAdsConn.nAmsPort,
	bExecute			:= ,
	sNetId				:= stAdsConn.sAmsNetId,
	ObjectType			:= F_BACnet_GetObjType(tObjectID),
	PropertyID			:= BACnetPropertyIdentifier_RecipientList,
	DataType			:= BACnetDataType_RecipientArr,
	ObjectInstance		:= F_BACnet_GetObjInstance(tObjectID),
	ptrValue			:= ADR(stBACnet_AdsBuffer.arrData),
	nLenValue			:= SIZEOF(stBACnet_AdsBuffer.arrData),
	bDone				=> ,
	bBusy				=> ,
	bError				=> ,
	nErrID				=> ,
	nProcessedLen		=> );

